# B&R Automation Studio project Embraco_LinkaNaOdlievanieRotorov_DokoncovaciaStanica_Rev2 (part 4)

#### OvladanieGripra.st
```iecst
ACTION OvladanieGripra:

	//Volanie funkcie SequenceControl//
	SequenceControl(SC:= SC_OvlGripra);

	CASE SC_OvlGripra.Step OF

		0:
			SC_OvlGripra.StepName:= '0 - Nulovanie';
			Otvor_Griper:= FALSE;
			Zatvor_Griper:= FALSE;
			doValcovanie_GriperOTVOR:= FALSE;
			doValcovanie_GriperZATVOR:= FALSE;
			IF SC_Valcovanie.Step <> 0 THEN
				SC_OvlGripra.ResetStep:= TRUE;
				SC_OvlGripra.Step:= 1;
			END_IF

		1:
			SC_OvlGripra.StepName:= '1 - Rozhodnutie o cinnosti';
			IF Otvor_Griper THEN
				SC_OvlGripra.Step:= 10;
			ELSIF Zatvor_Griper THEN
				SC_OvlGripra.Step:= 20;
			END_IF

		10:
			SC_OvlGripra.StepName:= '10 - Otvorenie gripra';
			SC_OvlGripra.IdleTime.PT:= T#3s;
			SC_OvlGripra.AlarmTime.PT:= T#3s;

			IF Valcovanie_Manual THEN
				SC_OvlGripra.IdleTime.IN:= TRUE;
			ELSE
				SC_OvlGripra.AlarmTime.IN:= TRUE;
			END_IF

			IF NOT SC_OvlGripra.Switch1 THEN
				doValcovanie_GriperOTVOR:= TRUE;
				SC_OvlGripra.Switch1:= TRUE;
			END_IF

			IF SC_OvlGripra.AlarmTime.Q THEN
				Alarmy[63]:= TRUE;
				PoruchaStanicaValcovania:= TRUE;
			END_IF

			IF diValcovanie_GriperOtvoreny OR SC_OvlGripra.IdleTime.Q THEN
				SC_OvlGripra.ResetStep:= TRUE;
				SC_OvlGripra.Step:= 0;
			END_IF

		20:
			SC_OvlGripra.StepName:= '20 - Zatvorenie gripra';
			SC_OvlGripra.IdleTime.PT:= T#3s;
			SC_OvlGripra.AlarmTime.PT:= T#3s;

			IF Valcovanie_Manual THEN
				SC_OvlGripra.IdleTime.IN:= TRUE;
			ELSE
				SC_OvlGripra.AlarmTime.IN:= TRUE;
			END_IF

			IF NOT SC_OvlGripra.Switch1 THEN
				doValcovanie_GriperZATVOR:= TRUE;
				SC_OvlGripra.Switch1:= TRUE;
			END_IF

			IF SC_OvlGripra.AlarmTime.Q THEN
				Alarmy[62]:= TRUE;
				PoruchaStanicaValcovania:= TRUE;
			END_IF

			IF diValcovanie_GriperZatvoreny OR SC_OvlGripra.IdleTime.Q THEN
				SC_OvlGripra.ResetStep:= TRUE;
				SC_OvlGripra.Step:= 0;
			END_IF

	END_CASE

			END_ACTION
```

#### OvladanieZdvihuRotora.st
```iecst
ACTION OvladanieZdvihuRotora:

	//Volanie funkcie SequenceControl//
	SequenceControl(SC:= SC_OvlZdvihu);

	CASE SC_OvlZdvihu.Step OF

		0:
			SC_OvlZdvihu.StepName:= '0 - Nulovanie';
			Rotor_ZDVIHNI:= FALSE;
			Rotor_POLOZ:= FALSE;
			doValcovanie_ZDVIH_Rotora:= FALSE;
			doValcovanie_ZOSTUP_Rotora:= FALSE;
			IF SC_Valcovanie.Step <> 0 THEN
				SC_OvlZdvihu.ResetStep:= TRUE;
				SC_OvlZdvihu.Step:= 1;
			END_IF

		1:
			SC_OvlZdvihu.StepName:= '1 - Rozhodnutie o cinnosti';
			IF Rotor_ZDVIHNI THEN
				SC_OvlZdvihu.Step:= 10;
			ELSIF Rotor_POLOZ THEN
				SC_OvlZdvihu.Step:= 20;
			END_IF

		10:
			SC_OvlZdvihu.StepName:= '10 - Zodvihnutie rotora';
			SC_OvlZdvihu.IdleTime.PT:= T#3s;
			SC_OvlZdvihu.AlarmTime.PT:= T#3s;

			IF Valcovanie_Manual THEN
				SC_OvlZdvihu.IdleTime.IN:= TRUE;
			ELSE
				SC_OvlZdvihu.AlarmTime.IN:= TRUE;
			END_IF

			IF NOT SC_OvlZdvihu.Switch1 THEN
				doValcovanie_ZDVIH_Rotora:= TRUE;
				SC_OvlZdvihu.Switch1:= TRUE;
			END_IF

			IF SC_OvlZdvihu.AlarmTime.Q THEN
				Alarmy[60]:= TRUE;
				PoruchaStanicaValcovania:= TRUE;
			END_IF

			IF diValcovanie_ZdvihHornaPoloha OR SC_OvlZdvihu.IdleTime.Q THEN
				SC_OvlZdvihu.ResetStep:= TRUE;
				SC_OvlZdvihu.Step:= 0;
			END_IF

		20:
			SC_OvlZdvihu.StepName:= '20 - Polozenie rotora';
			SC_OvlZdvihu.IdleTime.PT:= T#3s;
			SC_OvlZdvihu.AlarmTime.PT:= T#3s;

			IF Valcovanie_Manual THEN
				SC_OvlZdvihu.IdleTime.IN:= TRUE;
			ELSE
				SC_OvlZdvihu.AlarmTime.IN:= TRUE;
			END_IF

			IF NOT SC_OvlZdvihu.Switch1 THEN
				doValcovanie_ZOSTUP_Rotora:= TRUE;
				SC_OvlZdvihu.Switch1:= TRUE;
			END_IF

			IF SC_OvlZdvihu.AlarmTime.Q THEN
				Alarmy[61]:= TRUE;
				PoruchaStanicaValcovania:= TRUE;
			END_IF

			IF diValcovanie_ZdvihSpodnaPoloha OR SC_OvlZdvihu.IdleTime.Q THEN
				SC_OvlZdvihu.ResetStep:= TRUE;
				SC_OvlZdvihu.Step:= 0;
			END_IF

	END_CASE

			END_ACTION
```

#### OvladanieOtacaniaRotora.st
```iecst
ACTION OvladanieOtacaniaRotora:

	//Zadanie rýchlosti otáčania rotora//
	Valcovanie_FM_RychlostOtac_Hz:= TP_Valcovanie_RychlostOtacania;

	//Volanie funkcie SequenceControl//
	SequenceControl(SC:= SC_OvlOtacania);

	CASE SC_OvlOtacania.Step OF

		0:
			SC_OvlOtacania.StepName:= '0 - Nulovanie';
			FM_Menic[2].Input.Command.RunForward:= FALSE;
			FM_Menic[2].Input.Command.RunBackward:= FALSE;
			RotorOtacaj_VPRED:= FALSE;
			RotorOtacaj_VZAD:= FALSE;
			IF SC_Valcovanie.Step <> 0 THEN
				SC_OvlOtacania.ResetStep:= TRUE;
				SC_OvlOtacania.Step:= 1;
			END_IF

		1:
			SC_OvlOtacania.StepName:= '1 - Rozhodnutie o cinnosti';
			IF RotorOtacaj_VPRED THEN
				SC_OvlOtacania.Step:= 10;
			ELSIF RotorOtacaj_VZAD THEN
				SC_OvlOtacania.Step:= 20;
			END_IF

		10:
			SC_OvlOtacania.StepName:= '10 - Otacanie rotora VPRED';
			SC_OvlOtacania.IdleTime.PT:= T#5s;
			SC_OvlOtacania.AlarmTime.PT:= T#15s;
			FM_Menic[2].Input.HighSpeed:= (Valcovanie_FM_RychlostOtac_Hz * 10); //v Hz
			FM_Menic[2].Input.AccTime:= 1;  //0.1s
			FM_Menic[2].Input.DecTime:= 1;  //0.1s
			RotorOtacaj_VZAD:= FALSE;

			IF NOT SC_OvlOtacania.Switch1 THEN
				FM_Menic[2].Input.Command.RunForward:= TRUE;
				SC_OvlOtacania.Switch1:= TRUE;
			END_IF

			IF NOT RotorOtacaj_VPRED THEN
				SC_OvlOtacania.ResetStep:= TRUE;
				SC_OvlOtacania.Step:= 0;
			END_IF

		20:
			SC_OvlOtacania.StepName:= '20 - Otacanie rotora VZAD';
			SC_OvlOtacania.IdleTime.PT:= T#5s;
			SC_OvlOtacania.AlarmTime.PT:= T#15s;
			FM_Menic[2].Input.HighSpeed:= (Valcovanie_FM_RychlostOtac_Hz * 10); //v Hz
			FM_Menic[2].Input.AccTime:= 1;  //0.1s
			FM_Menic[2].Input.DecTime:= 1;  //0.1s
			RotorOtacaj_VPRED:= FALSE;

			IF NOT SC_OvlOtacania.Switch1 THEN
				FM_Menic[2].Input.Command.RunBackward:= TRUE;
				SC_OvlOtacania.Switch1:= TRUE;
			END_IF

			IF NOT RotorOtacaj_VZAD THEN
				SC_OvlOtacania.ResetStep:= TRUE;
				SC_OvlOtacania.Step:= 0;
			END_IF

	END_CASE

END_ACTION
```

### Program Logical/Program/StanicaVonkajsiehoValcovania (IEC)

#### Main.st - Init, cyclic, exit code
```iecst
PROGRAM _INIT
	(* Insert code here *)

END_PROGRAM

PROGRAM _CYCLIC

	//Volanie podprogramov//
	OvlHornehoPritlaku;
	OvlOtacaniaNastroja;
	OvlZdvihuRotora;

	//Volanie funkcie SequenceControl//
	SequenceControl(SC:= SC_Valcovanie2);

	Valcovanie2_CasStrekuOleja_s;
	Valcovanie2_CasValcovania_s;

	//***************************Dávka oleja**********************************//
	IF Valcovanie2_DavkaOleja THEN
		doValc2_DavkaOleja:= TRUE;
		CasDavkyOleja.IN:= TRUE;
	END_IF

	IF CasDavkyOleja.Q THEN
		Valcovanie2_DavkaOleja:= FALSE;
		CasDavkyOleja.IN:= FALSE;
		doValc2_DavkaOleja:= FALSE;
	END_IF

	CasDavkyOleja.PT:= REAL_TO_TIME(Valcovanie2_CasStrekuOleja_s * 1000);
	CasDavkyOleja();

	//Reset sekcie //
	IF Valcovanie2_Reset OR NOT BezpOkruhOplotenia_Aktivovany OR PoruchaStanicaValcovania2 THEN
		SC_Valcovanie2.Step:= 0;
	END_IF

	CASE SC_Valcovanie2.Step OF

		0:
			SC_Valcovanie2.StepName:='0 - Nulovanie';
			SC_OvlHornehoPritlaku.Step:= 0;
			SC_OvlOtacaniaNastroja.Step:= 0;
			SC_OvlZdvihuRotora.Step:= 0;
			Valcovanie2_Automat:= FALSE;
			Valcovanie2_KoniecVyroby:= FALSE;
			Valcovanie2_KoniecCyklu:= FALSE;
			Valcovanie2_Manual:= FALSE;
			Valcovanie2_PoINIT:= FALSE;
			Valcovanie2_Reset:= FALSE;
			Valcovanie2_ZdvihVPOZICI:= FALSE;
			Valcovanie2_UkoncilCyklus:= FALSE;
			RR_ZdvihRotora_PozValcovania:= FALSE;
			RR_ZdvihRotora_PozVychodzia:= FALSE;
			PocetCyklovValcovania:= 0;
			Priznak_ValcovanieNG:= FALSE;
			Priznak_ValcovanieOK:= FALSE;
			IF BezpOkruhOplotenia_Aktivovany AND NOT PoruchaStanicaValcovania2 THEN
				SC_Valcovanie2.ResetStep:= TRUE;
				SC_Valcovanie2.Step:= 1;
			END_IF

		1:
			SC_Valcovanie2.StepName:='1 - Rozhodnutie o cinnosti';
			IF Valcovanie2_Automat THEN
				SC_Valcovanie2.Step:= 2;
			ELSIF Valcovanie2_Manual THEN
				SC_Valcovanie2.Step:= 700;
			END_IF

			//********************************************************Inicializácia****************************************************************************//

		2:
			SC_Valcovanie2.StepName:='2 - Inicializacia - cakanie na spustenie';
			SC_Valcovanie2.IdleTime.PT:= T#500ms;
			SC_Valcovanie2.AlarmTime.PT:= T#5s;
			SC_Valcovanie2.IdleTime.IN:= TRUE;

			IF SC_Valcovanie2.IdleTime.Q AND diStol_SnimacPolohyStola THEN
				SC_Valcovanie2.ResetStep:= TRUE;
				SC_Valcovanie2.Step:= 4;
			END_IF

		4:
			SC_Valcovanie2.StepName:='4 - Inicializacia - kontrola home serva zdvihu rotora';
			SC_Valcovanie2.IdleTime.PT:= T#500ms;
			SC_Valcovanie2.AlarmTime.PT:= T#5s;

			IF Motion[4].status.DriveStatus.HomingOk THEN
				SC_Valcovanie2.ResetStep:= TRUE;
				SC_Valcovanie2.Step:= 6;
			ELSE
				SC_Valcovanie2.ResetStep:= TRUE;
				SC_Valcovanie2.Step:= 5;
			END_IF

		5:
			SC_Valcovanie2.StepName:='5 - Inicializacia - homing serva zdvihu rotora';
			SC_Valcovanie2.IdleTime.PT:= T#500ms;
			SC_Valcovanie2.AlarmTime.PT:= T#5s;

			IF NOT SC_Valcovanie2.Switch1 THEN
				ZdvihRotora_HOME:= TRUE;
				SC_Valcovanie2.Switch1:= TRUE;
			END_IF

			IF Motion[4].status.DriveStatus.HomingOk THEN
				SC_Valcovanie2.IdleTime.IN:= TRUE;
			END_IF

			IF Motion[4].status.DriveStatus.HomingOk AND SC_Valcovanie2.IdleTime.Q AND Motion[4].state.StandStill THEN
				SC_Valcovanie2.ResetStep:= TRUE;
				SC_Valcovanie2.Step:= 6;
			END_IF

		6:
			SC_Valcovanie2.StepName:='6 - Inicializacia - zasunutie zdvihu rotora do vychodiskovej pozicie';
			SC_Valcovanie2.IdleTime.PT:= T#500ms;
			SC_Valcovanie2.AlarmTime.PT:= T#5s;

			IF NOT SC_Valcovanie2.Switch1 AND (Valcovanie2_AktualPozMM <> Valcovanie2_ZadanaPozSTART_MM) AND SC_OvlZdvihuRotora.Step = 1 THEN
				ZdvihRotora_PoziciaSTART:= TRUE;
				SC_Valcovanie2.Switch1:= TRUE;
			END_IF

			IF (Valcovanie2_AktualPozMM = Valcovanie2_ZadanaPozSTART_MM) AND Motion[4].state.StandStill THEN
				SC_Valcovanie2.ResetStep:= TRUE;
				SC_Valcovanie2.Step:= 9;
			END_IF

		9:
			SC_Valcovanie2.StepName:='9 - Inicializacia - vysunutie horneho pritlaku dole';
			SC_Valcovanie2.IdleTime.PT:= T#4s;
			SC_Valcovanie2.AlarmTime.PT:= T#5s;

			IF NOT SC_Valcovanie2.Switch1 AND SC_OvlHornehoPritlaku.Step = 1 THEN
				HornyPritlak_DOLE:= TRUE;
				SC_Valcovanie2.Switch1:= TRUE;
			END_IF

			IF diValc2_PritlakVysunuty THEN
				SC_Valcovanie2.ResetStep:= TRUE;
				SC_Valcovanie2.Step:= 10;
			END_IF

		10:
			SC_Valcovanie2.StepName:='10 - Inicializacia - spustenie otacania nastroja';
			SC_Valcovanie2.IdleTime.PT:= T#4s;
			SC_Valcovanie2.AlarmTime.PT:= T#5s;

			IF NOT SC_Valcovanie2.Switch1 AND SC_OvlOtacaniaNastroja.Step = 1 AND VonkajsieValcovanie_AKTIVNE THEN
				OtacanieNastroja_VPRED:= TRUE;
				SC_Valcovanie2.IdleTime.IN:= TRUE;
				SC_Valcovanie2.Switch1:= TRUE;
			END_IF

			IF SC_Valcovanie2.IdleTime.Q OR NOT VonkajsieValcovanie_AKTIVNE THEN
				Valcovanie2_PoINIT:= TRUE;
				SC_Valcovanie2.ResetStep:= TRUE;
				SC_Valcovanie2.Step:= 100;
			END_IF

			//********************************************************Automatický režim****************************************************************************//
		100:
			SC_Valcovanie2.StepName:='100 - Automaticky rezim - cakanie na start cyklu';
			SC_Valcovanie2.IdleTime.PT:= T#500ms;
			SC_Valcovanie2.AlarmTime.PT:= T#5s;

            SC_Valcovanie2.IdleTime.IN:= NOT diValc2_PritomnostRotora;

			IF Valcovanie2_KoniecCyklu THEN
				SC_Valcovanie2.ResetStep:= TRUE;
				SC_Valcovanie2.Step:= 105;
			ELSIF NOT VonkajsieValcovanie_AKTIVNE THEN
				SC_Valcovanie2.ResetStep:= TRUE;
				SC_Valcovanie2.Step:= 120;
			ELSIF Stol_PoINIT AND NOT Valcovanie2_UkoncilCyklus AND diValc2_PritomnostRotora AND diStol_SnimacPolohyStola THEN
				SC_Valcovanie2.ResetStep:= TRUE;
				SC_Valcovanie2.Step:= 101;
			ELSIF Stol_PoINIT AND NOT Valcovanie2_UkoncilCyklus AND NOT diValc2_PritomnostRotora AND SC_Valcovanie2.IdleTime.Q THEN
				SC_Valcovanie2.ResetStep:= TRUE;
				SC_Valcovanie2.Step:= 120;
			ELSIF Valcovanie2_KoniecVyroby AND NOT Stol_Automat THEN
				SC_Valcovanie2.ResetStep:= TRUE;
				SC_Valcovanie2.Step:= 105;
			END_IF

		101:
			SC_Valcovanie2.StepName:='101 - Automaticky rezim - zdvih rotora, streknutie oleja';
			SC_Valcovanie2.IdleTime.PT:= T#500ms;
			SC_Valcovanie2.AlarmTime.PT:= T#5s;

			IF NOT SC_Valcovanie2.Switch1 AND SC_OvlZdvihuRotora.Step = 1 THEN
				ZdvihRotora_VALCOVANIE:= TRUE;
				SC_Valcovanie2.Switch1:= TRUE;
			END_IF

			IF Priznak_ValcovanieOK AND Valcovanie2_AktualPozMM = 13 AND Motion[4].state.StandStill AND diValc2_PritomnostRotora AND NOT diValc2_SpomalenieZdvihu THEN
				Priznak_ValcovanieOK:= FALSE;
				SC_Valcovanie2.ResetStep:= TRUE;
				SC_Valcovanie2.Step:= 120;
			ELSIF Priznak_ValcovanieOK AND Valcovanie2_AktualPozMM = 13 AND Motion[4].state.StandStill AND (NOT diValc2_PritomnostRotora OR diValc2_SpomalenieZdvihu) THEN
				Alarmy[74]:= TRUE;
				PoruchaStanicaValcovania2:= TRUE;
			ELSIF Priznak_ValcovanieNG AND (Valcovanie2_AktualPozMM = 13) AND Motion[4].state.StandStill THEN
				SC_Valcovanie2.ResetStep:= TRUE;
				SC_Valcovanie2.Step:= 110;
			END_IF

		105:
			SC_Valcovanie2.StepName:='105 - Automaticky rezim - zdvih vrchneho pritlaku';
			SC_Valcovanie2.IdleTime.PT:= T#500ms;
			SC_Valcovanie2.AlarmTime.PT:= T#5s;

			IF NOT SC_Valcovanie2.Switch1 THEN
				HornyPritlak_HORE:= TRUE;
			END_IF

			IF diValc2_PritlakZasunuty THEN
				SC_Valcovanie2.ResetStep:= TRUE;
				SC_Valcovanie2.Step:= 0;
			END_IF

		110:
			SC_Valcovanie2.StepName:='110 - Automaticky rezim - zdvih vrchneho pritlaku po NG kusu';
			SC_Valcovanie2.IdleTime.PT:= T#500ms;
			SC_Valcovanie2.AlarmTime.PT:= T#5s;

			IF NOT SC_Valcovanie2.Switch1 THEN
				HornyPritlak_HORE:= TRUE;
			END_IF

			IF diValc2_PritlakZasunuty THEN
				Alarmy[75]:= TRUE;
				PoruchaStanicaValcovania2:= TRUE;
			END_IF

		120:
			SC_Valcovanie2.StepName:='120 - Automaticky rezim - vystavenie signalu ukoncenie pracovneho cyklu';
			SC_Valcovanie2.IdleTime.PT:= T#500ms;
			SC_Valcovanie2.AlarmTime.PT:= T#5s;

			Valcovanie2_UkoncilCyklus:= TRUE;
			SC_Valcovanie2.ResetStep:= TRUE;
			SC_Valcovanie2.Step:= 121;

		121:
			SC_Valcovanie2.StepName:='121 - Automaticky rezim - cakanie na otocenie stola';
			SC_Valcovanie2.IdleTime.PT:= T#500ms;
			SC_Valcovanie2.AlarmTime.PT:= T#5s;

			IF NOT Valcovanie2_UkoncilCyklus THEN
				SC_Valcovanie2.ResetStep:= TRUE;
				SC_Valcovanie2.Step:= 100;
			ELSIF Valcovanie2_KoniecVyroby AND NOT Stol_Automat THEN
				SC_Valcovanie2.ResetStep:= TRUE;
				SC_Valcovanie2.Step:= 105;
			ELSIF Valcovanie2_KoniecCyklu THEN
				SC_Valcovanie2.ResetStep:= TRUE;
				SC_Valcovanie2.Step:= 105;
			END_IF

			//********************************************************Ručný režim***********************************************************************************//
		700:
			SC_Valcovanie2.StepName:='700 - Rucny rezim';

	END_CASE

				END_PROGRAM

PROGRAM _EXIT
				(* Insert code here *)

				END_PROGRAM
```

#### Variables.var - Local variables
```iecst
VAR
	SC_OvlZdvihuRotora : SequenceControlTyp;
	ZdvihRotora_JoggHORE : BOOL;
	ZdvihRotora_JoggDOLE : BOOL;
	ZdvihRotora_VALCOVANIE : BOOL;
	ZdvihRotora_HOME : BOOL;
	ZdvihRotora_PoziciaSTART : BOOL;
	ZdvihRotora_PoziciaVALCOVANIA : BOOL;
	SC_OvlOtacaniaNastroja : SequenceControlTyp;
	OtacanieNastroja_VPRED : BOOL;
	OtacanieNastroja_VZAD : BOOL;
	SC_OvlHornehoPritlaku : SequenceControlTyp;
	HornyPritlak_HORE : BOOL;
	HornyPritlak_DOLE : BOOL;
	CasDavkyOleja : TON;
	RR_ZdvihRotora_PozVychodzia : BOOL;
	RR_ZdvihRotora_PozValcovania : BOOL;
	PocetCyklovValcovania : USINT;
	Priznak_ValcovanieNG : BOOL;
	Priznak_ValcovanieOK : BOOL;
	TaktTime : TON;
	NameranyTaktime : TIME;
END_VAR
```

#### OvlZdvihuRotora.st
```iecst
ACTION OvlZdvihuRotora:

	//Parametre zdvihu rotora//
	Valcovanie2_ServoJoggRychl_MM_s;
	Valcovanie2_ServoPracRychl1_MM_s; //Rýchlost priblíženia
	Valcovanie2_ServoPracRychl2_MM_s; //Rýchlosť valcovania
	Valcovanie2_FM_RozbehRampa_s;
	Valcovanie2_FM_DobehRampa_s;
	Valcovanie2_MomentPritlaku_Nm:= 3; //3Nm

	//Volanie funkcie SequenceControl//
	SequenceControl(SC:= SC_OvlZdvihuRotora);

	CASE SC_OvlZdvihuRotora.Step OF

		0:
			SC_OvlZdvihuRotora.StepName:= '0 - Nulovanie';
			ZdvihRotora_JoggDOLE:= FALSE;
			ZdvihRotora_JoggHORE:= FALSE;
			ZdvihRotora_HOME:= FALSE;
			ZdvihRotora_VALCOVANIE:= FALSE;
			ZdvihRotora_PoziciaSTART:= FALSE;
			ZdvihRotora_PoziciaVALCOVANIA:= FALSE;
			Motion[4].cmd.home:= FALSE;
			Motion[4].cmd.moveAbsolute:= FALSE;
			Motion[4].cmd.moveJogNeg:= FALSE;
			Motion[4].cmd.moveJogPos:= FALSE;
			Motion[4].cmd.moveVelocity:= FALSE;
			Valcovanie2_PrebiehaHoming:= FALSE;
			Motion[4].par.direction:= 0;

			IF SC_Valcovanie2.Step <> 0 AND (NOT Motion[4].status.DriveStatus.HomingOk OR Motion[4].state.StandStill) THEN
				Motion[4].cmd.halt:= FALSE;
				SC_OvlZdvihuRotora.ResetStep:= TRUE;
				SC_OvlZdvihuRotora.Step:= 1;
			END_IF

		1:
			SC_OvlZdvihuRotora.StepName:= '1 - Rozhodnutie o cinnosti';
			IF ZdvihRotora_JoggDOLE THEN
				SC_OvlZdvihuRotora.Step:= 10;
			ELSIF ZdvihRotora_JoggHORE THEN
				SC_OvlZdvihuRotora.Step:= 20;
			ELSIF ZdvihRotora_HOME THEN
				SC_OvlZdvihuRotora.Step:= 30;
			ELSIF ZdvihRotora_VALCOVANIE THEN
				SC_OvlZdvihuRotora.Step:= 40;
			ELSIF ZdvihRotora_PoziciaSTART THEN
				SC_OvlZdvihuRotora.Step:= 50;
			ELSIF ZdvihRotora_PoziciaVALCOVANIA THEN
				SC_OvlZdvihuRotora.Step:= 60;
			END_IF

		10:
			SC_OvlZdvihuRotora.StepName:= '10 - Jogging DOLE';
			SC_OvlZdvihuRotora.IdleTime.PT:= T#3s;
			SC_OvlZdvihuRotora.AlarmTime.PT:= T#3s;

			Motion[4].par.velocityJog:= (Valcovanie2_ServoJoggRychl_MM_s * 100);
			Motion[4].par.acc := (Valcovanie2_ServoJoggRychl_MM_s * 1000);
			Motion[4].par.dec := (Valcovanie2_ServoJoggRychl_MM_s * 1000);

			IF NOT SC_OvlZdvihuRotora.Switch1 THEN
				Motion[4].cmd.moveJogNeg:= TRUE;
				SC_OvlZdvihuRotora.Switch1:= TRUE;
			END_IF

			IF (NOT ZdvihRotora_JoggDOLE OR Valcovanie2_AktualPozMM <= 13)THEN
				Motion[4].cmd.moveJogNeg:= FALSE;
				SC_OvlZdvihuRotora.ResetStep:= TRUE;
				SC_OvlZdvihuRotora.Step:= 0;
			END_IF

			IF diValc2_ZdvihSpodnyLimit THEN
				Motion[4].cmd.halt:= TRUE;
				Alarmy[56]:= TRUE;
				PoruchaStanicaValcovania2:= TRUE;
			END_IF

		20:
			SC_OvlZdvihuRotora.StepName:= '20 - Jogging HORE';
			SC_OvlZdvihuRotora.IdleTime.PT:= T#3s;
			SC_OvlZdvihuRotora.AlarmTime.PT:= T#3s;

			Motion[4].par.velocityJog:= (Valcovanie2_ServoJoggRychl_MM_s * 100);
			Motion[4].par.acc := (Valcovanie2_ServoJoggRychl_MM_s * 1000);
			Motion[4].par.dec := (Valcovanie2_ServoJoggRychl_MM_s * 1000);

			IF NOT SC_OvlZdvihuRotora.Switch1 THEN
				Motion[4].cmd.moveJogPos:= TRUE;
				SC_OvlZdvihuRotora.Switch1:= TRUE;
			END_IF

			IF (NOT ZdvihRotora_JoggHORE OR Valcovanie2_AktualPozMM >= 185)THEN
				Motion[4].cmd.moveJogPos:= FALSE;
				SC_OvlZdvihuRotora.ResetStep:= TRUE;
				SC_OvlZdvihuRotora.Step:= 0;
			END_IF

			IF diValc2_ZdvihHornyLimit THEN
				Motion[4].cmd.halt:= TRUE;
				Alarmy[56]:= TRUE;
				PoruchaStanicaValcovania2:= TRUE;
			END_IF

		30:
			SC_OvlZdvihuRotora.StepName:= '30 - Start homingu';
			SC_OvlZdvihuRotora.IdleTime.PT:= T#500ms;
			SC_OvlZdvihuRotora.AlarmTime.PT:= T#3s;

			IF NOT SC_OvlZdvihuRotora.Switch1 THEN
				Motion[4].cmd.home:= TRUE;
				Valcovanie2_PrebiehaHoming:= TRUE;
				SC_OvlZdvihuRotora.IdleTime.IN:= TRUE;
				SC_OvlZdvihuRotora.Switch1:= TRUE;
			END_IF

			IF SC_OvlZdvihuRotora.IdleTime.Q THEN
				SC_OvlZdvihuRotora.ResetStep:= TRUE;
				SC_OvlZdvihuRotora.Step:= 31;
			END_IF

		31:
			SC_OvlZdvihuRotora.StepName:= '31 - Ukoncenie homingu';
			SC_OvlZdvihuRotora.IdleTime.PT:= T#3s;
			SC_OvlZdvihuRotora.AlarmTime.PT:= T#3s;

			IF Valcovanie2_HomingOK AND Motion[4].state.StandStill THEN
				SC_OvlZdvihuRotora.ResetStep:= TRUE;
				SC_OvlZdvihuRotora.Step:= 0;
			END_IF

		40:
			SC_OvlZdvihuRotora.StepName:= '40 - Valcovanie,chod rychlo na spomalovaci snimac';
			SC_OvlZdvihuRotora.IdleTime.PT:= T#3s;
			SC_OvlZdvihuRotora.AlarmTime.PT:= T#3s;

			Motion[4].par.velocity:= (Valcovanie2_ServoPracRychl1_MM_s * 100);
			Motion[4].par.acc := (Valcovanie2_ServoPracRychl1_MM_s * 1000);
			Motion[4].par.dec := (Valcovanie2_ServoPracRychl1_MM_s * 1000);
			Motion[4].par.direction:= 0;

			IF NOT SC_OvlZdvihuRotora.Switch1 THEN
				Motion[4].cmd.moveVelocity:= TRUE;
				PocetCyklovValcovania:= PocetCyklovValcovania + 1;
				TaktTime.IN:= TRUE;
				SC_OvlZdvihuRotora.Switch1:= TRUE;
			END_IF

			IF EDGEPOS(diValc2_SpomalenieZdvihu) THEN
				SC_OvlZdvihuRotora.ResetStep:= TRUE;
				SC_OvlZdvihuRotora.Step:= 41;
			ELSIF Valcovanie2_AktualPozMM >= 118 THEN
				SC_OvlZdvihuRotora.ResetStep:= TRUE;
				SC_OvlZdvihuRotora.Step:= 41;
			ELSIF diValc2_ZdvihHornyLimit THEN
				Motion[4].cmd.halt:= TRUE;
				Alarmy[56]:= TRUE;
				PoruchaStanicaValcovania2:= TRUE;
			END_IF

		41:
			SC_OvlZdvihuRotora.StepName:= '41 - Valcovanie,chod pomaly na poziciu';
			SC_OvlZdvihuRotora.IdleTime.PT:= T#1s;
			SC_OvlZdvihuRotora.AlarmTime.PT:= T#3s;

			Motion[4].par.velocity:= (Valcovanie2_ServoPracRychl2_MM_s * 100);
			Motion[4].par.acc := (Valcovanie2_ServoPracRychl2_MM_s * 1000);
			Motion[4].par.dec := (Valcovanie2_ServoPracRychl2_MM_s * 1000);
			Motion[4].par.position:= (Valcovanie2_ZadanaPozMM * 100); //180mm

			IF NOT SC_OvlZdvihuRotora.Switch1 THEN
				Motion[4].cmd.moveAbsolute:= TRUE;
				IF PocetCyklovValcovania >= Valcovanie2_PocetCyklStrekuOleja THEN
					Valcovanie2_DavkaOleja:= TRUE;
					PocetCyklovValcovania:= 0;
				END_IF
				SC_OvlZdvihuRotora.Switch1:= TRUE;
			END_IF

			IF (Valcovanie2_AktualPozMM = Valcovanie2_ZadanaPozMM) AND Motion[4].state.StandStill THEN
				SC_OvlZdvihuRotora.ResetStep:= TRUE;
				SC_OvlZdvihuRotora.Step:= 45;
			ELSIF Motion[4].status.ActTorque >= 20 THEN
				Motion[4].cmd.halt:= TRUE;
				Priznak_ValcovanieNG:= TRUE;
				SC_OvlZdvihuRotora.ResetStep:= TRUE;
				SC_OvlZdvihuRotora.Step:= 42;
			ELSIF diValc2_ZdvihHornyLimit THEN
				Motion[4].cmd.halt:= TRUE;
				Alarmy[56]:= TRUE;
				PoruchaStanicaValcovania2:= TRUE;
			END_IF

		42:
			SC_OvlZdvihuRotora.StepName:= '42 - Valcovanie,zastavenie po dosiahnutí momentu';
			SC_OvlZdvihuRotora.IdleTime.PT:= T#1s;
			SC_OvlZdvihuRotora.AlarmTime.PT:= T#3s;
			SC_OvlZdvihuRotora.IdleTime.IN:= TRUE;

			IF NOT Motion[4].cmd.halt THEN
				SC_OvlZdvihuRotora.ResetStep:= TRUE;
				SC_OvlZdvihuRotora.Step:= 45;
			END_IF

			IF SC_OvlZdvihuRotora.IdleTime.Q THEN
				Motion[4].cmd.halt:= FALSE;
			END_IF

		45:
			SC_OvlZdvihuRotora.StepName:= '45 - Valcovanie,chod pomalou rychlostou dole';
			SC_OvlZdvihuRotora.IdleTime.PT:= T#50ms;
			SC_OvlZdvihuRotora.AlarmTime.PT:= T#3s;
			SC_OvlZdvihuRotora.IdleTime.IN:= TRUE;

			Motion[4].par.velocity:= (Valcovanie2_ServoPracRychl1_MM_s * 100);
			Motion[4].par.acc := (Valcovanie2_ServoPracRychl1_MM_s * 1000);
			Motion[4].par.dec := (Valcovanie2_ServoPracRychl1_MM_s * 1000);
			Motion[4].par.direction:= 1;

			IF NOT SC_OvlZdvihuRotora.Switch1 AND SC_OvlZdvihuRotora.IdleTime.Q THEN
				Motion[4].cmd.moveVelocity:= TRUE;
				SC_OvlZdvihuRotora.Switch1:= TRUE;
			END_IF

			IF NOT diValc2_SpomalenieZdvihu AND Valcovanie2_AktualPozMM < 118 THEN
				SC_OvlZdvihuRotora.ResetStep:= TRUE;
				SC_OvlZdvihuRotora.Step:= 46;
			ELSIF Valcovanie2_AktualPozMM <= 95 THEN
				SC_OvlZdvihuRotora.ResetStep:= TRUE;
				SC_OvlZdvihuRotora.Step:= 46;
			ELSIF diValc2_ZdvihSpodnyLimit THEN
				Motion[4].cmd.halt:= TRUE;
				Alarmy[56]:= TRUE;
				PoruchaStanicaValcovania2:= TRUE;
			END_IF

		46:
			SC_OvlZdvihuRotora.StepName:= '46 - Valcovanie, chod rychlo do vychodiskovej pozicie';
			SC_OvlZdvihuRotora.IdleTime.PT:= T#3s;
			SC_OvlZdvihuRotora.AlarmTime.PT:= T#3s;

			Motion[4].par.velocity:= (Valcovanie2_ServoPracRychl1_MM_s * 100);
			Motion[4].par.acc := (Valcovanie2_ServoPracRychl1_MM_s * 1000);
			Motion[4].par.dec := (Valcovanie2_ServoPracRychl1_MM_s * 1000);
			Motion[4].par.position:= 1300; //13mm

			IF NOT SC_OvlZdvihuRotora.Switch1 THEN
				Motion[4].cmd.moveAbsolute:= TRUE;
				SC_OvlZdvihuRotora.Switch1:= TRUE;
			END_IF

			IF (Valcovanie2_AktualPozMM = 13) AND Motion[4].state.StandStill AND NOT Priznak_ValcovanieNG THEN
				Priznak_ValcovanieOK:= TRUE;
				NameranyTaktime:= TaktTime.ET;
				TaktTime.IN:= FALSE;
				SC_OvlZdvihuRotora.ResetStep:= TRUE;
				SC_OvlZdvihuRotora.Step:= 0;
			ELSIF diValc2_ZdvihSpodnyLimit THEN
				Motion[4].cmd.halt:= TRUE;
				Alarmy[56]:= TRUE;
				PoruchaStanicaValcovania2:= TRUE;
			END_IF

		50:
			SC_OvlZdvihuRotora.StepName:= '50 - Presun do pozicie START';
			SC_OvlZdvihuRotora.IdleTime.PT:= T#3s;
			SC_OvlZdvihuRotora.AlarmTime.PT:= T#3s;

			Motion[4].par.velocity:= (Valcovanie2_ServoPracRychl1_MM_s * 100);
			Motion[4].par.acc := (Valcovanie2_ServoPracRychl1_MM_s * 1000);
			Motion[4].par.dec := (Valcovanie2_ServoPracRychl1_MM_s * 1000);
			Motion[4].par.position:= 1300; //13mm

			IF NOT SC_OvlZdvihuRotora.Switch1 THEN
				Motion[4].cmd.moveAbsolute:= TRUE;
				SC_OvlZdvihuRotora.Switch1:= TRUE;
			END_IF

			IF (Valcovanie2_AktualPozMM = 13) AND Motion[4].state.StandStill THEN
				Valcovanie2_ZdvihVPOZICI:= TRUE;
				SC_OvlZdvihuRotora.ResetStep:= TRUE;
				SC_OvlZdvihuRotora.Step:= 0;
			ELSIF diValc2_ZdvihSpodnyLimit THEN
				Motion[4].cmd.halt:= TRUE;
				Alarmy[56]:= TRUE;
				PoruchaStanicaValcovania2:= TRUE;
			END_IF

		60:
			SC_OvlZdvihuRotora.StepName:= '60 - Presun do pozicie VALCOVANIA';
			SC_OvlZdvihuRotora.IdleTime.PT:= T#3s;
			SC_OvlZdvihuRotora.AlarmTime.PT:= T#3s;

			Motion[4].par.velocity:= (Valcovanie2_ServoPracRychl2_MM_s * 100);
			Motion[4].par.acc := (Valcovanie2_ServoPracRychl2_MM_s * 1000);
			Motion[4].par.dec := (Valcovanie2_ServoPracRychl2_MM_s * 1000);
			Motion[4].par.position:= (Valcovanie2_ZadanaPozMM * 100); //180mm

			IF NOT SC_OvlZdvihuRotora.Switch1 THEN
				Motion[4].cmd.moveAbsolute:= TRUE;
				SC_OvlZdvihuRotora.Switch1:= TRUE;
			END_IF

			IF (Valcovanie2_AktualPozMM = Valcovanie2_ZadanaPozMM) AND Motion[4].state.StandStill THEN
				Valcovanie2_ZdvihVPOZICI:= TRUE;
				SC_OvlZdvihuRotora.ResetStep:= TRUE;
				SC_OvlZdvihuRotora.Step:= 0;
			ELSIF Motion[4].status.ActTorque >= 5 THEN
				Motion[4].cmd.halt:= TRUE;
				SC_OvlZdvihuRotora.ResetStep:= TRUE;
				SC_OvlZdvihuRotora.Step:= 0;
			ELSIF diValc2_ZdvihHornyLimit THEN
				Motion[4].cmd.halt:= TRUE;
				Alarmy[56]:= TRUE;
				PoruchaStanicaValcovania2:= TRUE;
			END_IF

	END_CASE

	TaktTime.PT:= T#20s;
	TaktTime();

END_ACTION
```

#### OvlOtacaniaNastroja.st
```iecst
ACTION OvlOtacaniaNastroja:

	//Volanie funkcie SequenceControl//
	SequenceControl(SC:= SC_OvlOtacaniaNastroja);

	CASE SC_OvlOtacaniaNastroja.Step OF

		0:
			SC_OvlOtacaniaNastroja.StepName:= '0 - Nulovanie';
			FM_Menic[3].Input.Command.RunForward:= FALSE;
			FM_Menic[3].Input.Command.RunBackward:= FALSE;
			OtacanieNastroja_VPRED:= FALSE;
			OtacanieNastroja_VZAD:= FALSE;
			TP_Valcovanie2_ZamkniOtacVPRED:= FALSE;
			TP_Valcovanie2_ZamkniOtacVZAD:= FALSE;
			IF SC_Valcovanie2.Step <> 0 THEN
				SC_OvlOtacaniaNastroja.ResetStep:= TRUE;
				SC_OvlOtacaniaNastroja.Step:= 1;
			END_IF

		1:
			SC_OvlOtacaniaNastroja.StepName:= '1 - Rozhodnutie o cinnosti';
			IF OtacanieNastroja_VPRED THEN
				SC_OvlOtacaniaNastroja.Step:= 10;
			ELSIF OtacanieNastroja_VZAD THEN
				SC_OvlOtacaniaNastroja.Step:= 20;
			END_IF

		10:
			SC_OvlOtacaniaNastroja.StepName:= '10 - Otacanie nastroja VPRED';
			SC_OvlOtacaniaNastroja.IdleTime.PT:= T#5s;
			SC_OvlOtacaniaNastroja.AlarmTime.PT:= T#3s;
			FM_Menic[3].Input.HighSpeed:= REAL_TO_INT(Valcovanie2_FM_RychlostOtac_Hz * 10); //v Hz
			FM_Menic[3].Input.AccTime:=  REAL_TO_UINT(Valcovanie2_FM_RozbehRampa_s * 10);  //4s
			FM_Menic[3].Input.DecTime:= REAL_TO_UINT(Valcovanie2_FM_DobehRampa_s * 10);  //4s

			IF NOT SC_OvlOtacaniaNastroja.Switch1 THEN
				FM_Menic[3].Input.Command.RunForward:= TRUE;
				TP_Valcovanie2_ZamkniOtacVZAD:= TRUE;
				SC_OvlOtacaniaNastroja.Switch1:= TRUE;
			END_IF

			IF NOT OtacanieNastroja_VPRED THEN
				FM_Menic[3].Input.Command.RunForward:= FALSE;
			END_IF

			IF NOT OtacanieNastroja_VPRED AND NOT FM_Menic[3].Output.Status.Running THEN
				SC_OvlOtacaniaNastroja.ResetStep:= TRUE;
				SC_OvlOtacaniaNastroja.Step:= 0;
			END_IF

		20:
			SC_OvlOtacaniaNastroja.StepName:= '20 - Otacanie nastroja VZAD';
			SC_OvlOtacaniaNastroja.IdleTime.PT:= T#5s;
			SC_OvlOtacaniaNastroja.AlarmTime.PT:= T#3s;
			FM_Menic[3].Input.HighSpeed:= REAL_TO_INT(Valcovanie2_FM_RychlostOtac_Hz * 10); //v Hz
			FM_Menic[3].Input.AccTime:=  REAL_TO_UINT(Valcovanie2_FM_RozbehRampa_s * 10);  //4s
			FM_Menic[3].Input.DecTime:= REAL_TO_UINT(Valcovanie2_FM_DobehRampa_s * 10);  //4s

			IF NOT SC_OvlOtacaniaNastroja.Switch1 THEN
				FM_Menic[3].Input.Command.RunBackward:= TRUE;
				TP_Valcovanie2_ZamkniOtacVPRED:= TRUE;
				SC_OvlOtacaniaNastroja.Switch1:= TRUE;
			END_IF

			IF NOT OtacanieNastroja_VZAD THEN
				FM_Menic[3].Input.Command.RunBackward:= FALSE;
			END_IF

			IF NOT OtacanieNastroja_VZAD AND NOT FM_Menic[3].Output.Status.Running THEN
				SC_OvlOtacaniaNastroja.ResetStep:= TRUE;
				SC_OvlOtacaniaNastroja.Step:= 0;
			END_IF

	END_CASE

			END_ACTION
```

#### OvlHornehoPritlaku.st
```iecst
ACTION OvlHornehoPritlaku:

	//Volanie funkcie SequenceControl//
	SequenceControl(SC:= SC_OvlHornehoPritlaku);

	CASE SC_OvlHornehoPritlaku.Step OF

		0:
			SC_OvlHornehoPritlaku.StepName:= '0 - Nulovanie';
			HornyPritlak_DOLE:= FALSE;
			HornyPritlak_HORE:= FALSE;
			doValc2_ZdvihPritlakuHORE:= FALSE;
//			doValcovanie2_ZostupPritlakuDOLE:= FALSE;
			IF SC_Valcovanie2.Step <> 0 THEN
				SC_OvlHornehoPritlaku.ResetStep:= TRUE;
				SC_OvlHornehoPritlaku.Step:= 1;
			END_IF

		1:
			SC_OvlHornehoPritlaku.StepName:= '1 - Rozhodnutie o cinnosti';
			IF HornyPritlak_HORE THEN
				SC_OvlHornehoPritlaku.Step:= 10;
			ELSIF HornyPritlak_DOLE THEN
				SC_OvlHornehoPritlaku.Step:= 20;
			END_IF

		10:
			SC_OvlHornehoPritlaku.StepName:= '10 - Zodvihnutie horneho pritlaku hore';
			SC_OvlHornehoPritlaku.IdleTime.PT:= T#3s;
			SC_OvlHornehoPritlaku.AlarmTime.PT:= T#3s;

			IF Valcovanie2_Manual THEN
				SC_OvlHornehoPritlaku.IdleTime.IN:= TRUE;
			ELSE
				SC_OvlHornehoPritlaku.AlarmTime.IN:= TRUE;
			END_IF

			IF NOT SC_OvlHornehoPritlaku.Switch1 THEN
				doValc2_ZostupPritlakuDOLE:= FALSE;
				doValc2_ZdvihPritlakuHORE:= TRUE;
				SC_OvlHornehoPritlaku.Switch1:= TRUE;
			END_IF

			IF SC_OvlHornehoPritlaku.AlarmTime.Q THEN
				Alarmy[57]:= TRUE;
				PoruchaStanicaValcovania2:= TRUE;
			END_IF

			IF diValc2_PritlakZasunuty OR SC_OvlHornehoPritlaku.IdleTime.Q THEN
				SC_OvlHornehoPritlaku.ResetStep:= TRUE;
				SC_OvlHornehoPritlaku.Step:= 0;
			END_IF

		20:
			SC_OvlHornehoPritlaku.StepName:= '20 - Zostup horneho pritlaku dole';
			SC_OvlHornehoPritlaku.IdleTime.PT:= T#3s;
			SC_OvlHornehoPritlaku.AlarmTime.PT:= T#3s;

			IF Valcovanie2_Manual THEN
				SC_OvlHornehoPritlaku.IdleTime.IN:= TRUE;
			ELSE
				SC_OvlHornehoPritlaku.AlarmTime.IN:= TRUE;
			END_IF

			IF NOT SC_OvlHornehoPritlaku.Switch1 THEN
				doValc2_ZdvihPritlakuHORE:= FALSE;
				doValc2_ZostupPritlakuDOLE:= TRUE;
				SC_OvlHornehoPritlaku.Switch1:= TRUE;
			END_IF

			IF SC_OvlHornehoPritlaku.AlarmTime.Q THEN
				Alarmy[58]:= TRUE;
				PoruchaStanicaValcovania2:= TRUE;
			END_IF

			IF diValc2_PritlakVysunuty OR SC_OvlHornehoPritlaku.IdleTime.Q THEN
				SC_OvlHornehoPritlaku.ResetStep:= TRUE;
				SC_OvlHornehoPritlaku.Step:= 0;
			END_IF

	END_CASE

END_ACTION
```

### Program Logical/Program/StanicaMerania (IEC)

#### Main.st - Init, cyclic, exit code
```iecst
PROGRAM _INIT
	(* Insert code here *)

END_PROGRAM

PROGRAM _CYCLIC

	diTlacitko_RotorNG;
	diTlacitko_RotorOK;
	doZelenaLED_Tlacitko_rotor_OK;
	doCervenaLED_Tlacitko_rotor_NG;
	diMeranie_Osciloskop_Stav_NG;
	diMeranie_Osciloskop_Stav_OK;
	doMeranie_Osciloskop_START;
	doMeranie_Osciloskop_STOP;

	//Ovládanie vzorkovacej frekvencie osciloskopu//
	IF RotorOtacaj_VPRED THEN
		doMeranie_Osciloskop_Frekvencia:= Blikac50ms;
	ELSE
		doMeranie_Osciloskop_Frekvencia:= FALSE;
	END_IF

	//Meranie prestoja na stanici merania//
	IF StratovyCas_START THEN
		StratovyCas_Milisekundy:= StratovyCas_Milisekundy + 1;
		IF StratovyCas_Milisekundy >= 1000 THEN
			StratovyCas_Sekundy:= StratovyCas_Sekundy + 1;
			StratovyCas_Milisekundy:= 0;
		END_IF
		IF StratovyCas_Sekundy >= 60 THEN
			StratovyCas_Minuty:= StratovyCas_Minuty + 1;
			StratovyCas_Sekundy:= 0;
		END_IF
		IF StratovyCas_Minuty >= 60 THEN
			StratovyCas_Hodiny:= StratovyCas_Hodiny + 1;
			StratovyCas_Minuty:= 0;
		END_IF
		IF StratovyCas_Hodiny >= 24 THEN
			StratovyCas_RESET:= TRUE;
		END_IF
	END_IF

	IF StratovyCas_RESET THEN
		StratovyCas_Milisekundy:= 0;
		StratovyCas_Sekundy:= 0;
		StratovyCas_Minuty:= 0;
		StratovyCas_Hodiny:= 0;
		StratovyCas_RESET:= FALSE;
	END_IF

	//Volanie podprogramov//
	OvladanieOtacaniaRotora;
	OvladanieZdvihu;

	//Volanie funkcie SequenceControl//
	SequenceControl(SC:= SC_Meranie);

	//Prepočet času merania//
	CasMerania:= REAL_TO_TIME(TP_Meranie_CasMerania*1000);

	//Reset sekcie //
	IF Meranie_Reset OR NOT BezpOkruhOplotenia_Aktivovany OR PoruchaStanicaMerania THEN
		SC_Meranie.Step:= 0;
	END_IF

	CASE SC_Meranie.Step OF

		0:
			SC_Meranie.StepName:='0 - Nulovanie';
			SC_OvlOtacania.Step:= 0;
			SC_OvlZdvihu.Step:= 0;;
			Meranie_Automat:= FALSE;
			Meranie_KoniecVyroby:= FALSE;
			Meranie_KoniecCyklu:= FALSE;
			Meranie_Manual:= FALSE;
			Meranie_PoINIT:= FALSE;
			Meranie_Reset:= FALSE;
			Meranie_UkoncilCyklus:= FALSE;
			Meranie_ObsluhaRozhodla:= FALSE;
			doCervenaLED_Tlacitko_rotor_NG:= FALSE;
			doZelenaLED_Tlacitko_rotor_OK:= FALSE;
			StratovyCas_START:= FALSE;
			doMeranie_Osciloskop_START:= FALSE;
			IF BezpOkruhOplotenia_Aktivovany AND NOT PoruchaStanicaMerania THEN
				SC_Meranie.ResetStep:= TRUE;
				SC_Meranie.Step:= 1;
			END_IF

		1:
			SC_Meranie.StepName:='1 - Rozhodnutie o cinnosti';
			IF Meranie_Automat THEN
				SC_Meranie.Step:= 2;
			ELSIF Meranie_Manual THEN
				SC_Meranie.Step:= 700;
			END_IF

			//********************************************************Inicializácia****************************************************************************//

		2:
			SC_Meranie.StepName:='2 - Inicializacia - cakanie na spustenie';
			SC_Meranie.IdleTime.PT:= T#500ms;
			SC_Meranie.AlarmTime.PT:= T#5s;
			SC_Meranie.IdleTime.IN:= TRUE;

			IF SC_Meranie.IdleTime.Q THEN
				SC_Meranie.ResetStep:= TRUE;
				SC_Meranie.Step:= 3;
			END_IF

		3:
			SC_Meranie.StepName:='2 - Inicializacia - zasunutie zdvihu rotora';
			SC_Meranie.IdleTime.PT:= T#500ms;
			SC_Meranie.AlarmTime.PT:= T#5s;

			IF NOT SC_Meranie.Switch1 THEN
				Rotor_POLOZ:= TRUE;
				SC_Meranie.Switch1:= TRUE;
			END_IF

			IF diMeranie_ZdvihSpodnaPoloha THEN
				RotorOtacaj_VPRED:= TRUE;
				Meranie_PoINIT:= TRUE;
				SC_Meranie.ResetStep:= TRUE;
				SC_Meranie.Step:= 100;
			END_IF

			//********************************************************Automatický režim****************************************************************************//
		100:
			SC_Meranie.StepName:='100 - Automaticky rezim - cakanie na start cyklu';
			SC_Meranie.IdleTime.PT:= T#500ms;
			SC_Meranie.AlarmTime.PT:= T#5s;

           SC_Meranie.IdleTime.IN:= NOT diMeranie_PritomnostRotora;

			IF Meranie_KoniecCyklu THEN
				SC_Meranie.ResetStep:= TRUE;
				SC_Meranie.Step:= 0;
			ELSIF Zariadenie_PrebiehaRevorkRezim THEN
				SC_Meranie.ResetStep:= TRUE;
				SC_Meranie.Step:= 120;
			ELSIF Stol_PoINIT AND NOT Meranie_UkoncilCyklus AND diMeranie_PritomnostRotora AND diStol_SnimacPolohyStola THEN
				Meranie_ObsluhaRozhodla:= FALSE;
				doCervenaLED_Tlacitko_rotor_NG:= FALSE;
				doZelenaLED_Tlacitko_rotor_OK:= FALSE;
				SC_Meranie.ResetStep:= TRUE;
				SC_Meranie.Step:= 101;
			ELSIF Stol_PoINIT AND NOT Meranie_UkoncilCyklus AND NOT diMeranie_PritomnostRotora AND SC_Meranie.IdleTime.Q THEN
				Meranie_ObsluhaRozhodla:= FALSE;
				doCervenaLED_Tlacitko_rotor_NG:= FALSE;
				doZelenaLED_Tlacitko_rotor_OK:= FALSE;
				Stol_Pozicia_1:= 0;
				SC_Meranie.ResetStep:= TRUE;
				SC_Meranie.Step:= 120;
			ELSIF Meranie_KoniecVyroby AND NOT Stol_Automat THEN
				SC_Meranie.ResetStep:= TRUE;
				SC_Meranie.Step:= 0;
			END_IF

		101:
			SC_Meranie.StepName:='101 - Automaticky rezim - zdvih rotora';
			SC_Meranie.IdleTime.PT:= T#1s;
			SC_Meranie.AlarmTime.PT:= T#5s;

			IF NOT SC_Meranie.Switch1 AND SC_OvlZdvihu.Step = 1 THEN
				Rotor_ZDVIHNI:= TRUE;
				SC_Meranie.IdleTime.IN:= TRUE;
				SC_Meranie.Switch1:= TRUE;
			END_IF

			IF diMeranie_ZdvihHornaPoloha THEN
				SC_Meranie.ResetStep:= TRUE;
				SC_Meranie.Step:= 102;
			END_IF

		102:
			SC_Meranie.StepName:='102 - Automaticky rezim - spustenie otacania, cakanie na vysledok merania';
			SC_Meranie.IdleTime.PT:= T#5s;
			SC_Meranie.AlarmTime.PT:= T#2s;
			SC_Meranie.IdleTime.IN:= TRUE;

			IF NOT SC_Meranie.Switch1 THEN
				RotorOtacaj_VPRED:= TRUE;
				doMeranie_Osciloskop_START:= TRUE;
				SC_Meranie.AlarmTime.IN:= TRUE;
				SC_Meranie.Switch1:= TRUE;
			END_IF

			IF SC_Meranie.IdleTime.Q THEN
				StratovyCas_START:= TRUE;
			END_IF

			IF EDGEPOS(diMeranie_Osciloskop_Stav_OK) THEN
				Stol_Pozicia_1:= 1;
				StratovyCas_START:= FALSE;
				doMeranie_Osciloskop_START:= FALSE;
				SC_Meranie.ResetStep:= TRUE;
				SC_Meranie.Step:= 103;
			ELSIF EDGEPOS(diMeranie_Osciloskop_Stav_NG) THEN
				Stol_Pozicia_1:= 2;
				StratovyCas_START:= FALSE;
				doMeranie_Osciloskop_START:= FALSE;
				SC_Meranie.ResetStep:= TRUE;
				SC_Meranie.Step:= 103;
			ELSIF Meranie_KoniecCyklu THEN
				StratovyCas_START:= FALSE;
				doMeranie_Osciloskop_START:= FALSE;
				SC_Meranie.ResetStep:= TRUE;
				SC_Meranie.Step:= 103;
			END_IF

		103:
			SC_Meranie.StepName:='103 - Automaticky rezim - zasunutie zdvihu rotora';
			SC_Meranie.IdleTime.PT:= T#5s;
			SC_Meranie.AlarmTime.PT:= T#5s;

			IF NOT SC_Meranie.Switch1  AND SC_OvlZdvihu.Step = 1 THEN
				Rotor_POLOZ:= TRUE;
				SC_Meranie.Switch1:= TRUE;
			END_IF

			IF diMeranie_ZdvihSpodnaPoloha AND diMeranie_PritomnostRotora AND NOT diMeranie_ZdvihHornaPoloha THEN
				SC_Meranie.ResetStep:= TRUE;
				SC_Meranie.Step:= 120;
			ELSIF diMeranie_ZdvihSpodnaPoloha AND NOT diMeranie_PritomnostRotora THEN
				Alarmy[73]:= TRUE;
				PoruchaStanicaMerania:= TRUE;
			ELSIF diMeranie_ZdvihSpodnaPoloha AND diMeranie_ZdvihHornaPoloha THEN
				Alarmy[73]:= TRUE;
				PoruchaStanicaMerania:= TRUE;
			END_IF

		120:
			SC_Meranie.StepName:='120 - Automaticky rezim - vystavenie signalu ukoncenie pracovneho cyklu';
			SC_Meranie.IdleTime.PT:= T#5s;
			SC_Meranie.AlarmTime.PT:= T#5s;

			Meranie_UkoncilCyklus:= TRUE;
			SC_Meranie.ResetStep:= TRUE;
			SC_Meranie.Step:= 121;

		121:
			SC_Meranie.StepName:='121 - Automaticky rezim - cakanie na otocenie stola';
			SC_Meranie.IdleTime.PT:= T#5s;
			SC_Meranie.AlarmTime.PT:= T#5s;

			IF NOT Meranie_UkoncilCyklus THEN
				SC_Meranie.ResetStep:= TRUE;
				SC_Meranie.Step:= 100;
			ELSIF Meranie_KoniecVyroby AND NOT Stol_Automat THEN
				SC_Meranie.ResetStep:= TRUE;
				SC_Meranie.Step:= 0;
			ELSIF Meranie_KoniecCyklu THEN
				SC_Meranie.ResetStep:= TRUE;
				SC_Meranie.Step:= 0;
			END_IF

			//********************************************************Ručný režim***********************************************************************************//
		700:
			SC_Meranie.StepName:='700 - Rucny rezim';

	END_CASE

				END_PROGRAM

PROGRAM _EXIT
				(* Insert code here *)

				END_PROGRAM
```

#### Variables.var - Local variables
```iecst
VAR
	SC_OvlZdvihu : SequenceControlTyp;
	Rotor_ZDVIHNI : BOOL;
	Rotor_POLOZ : BOOL;
	SC_OvlOtacania : SequenceControlTyp;
	RotorOtacaj_VPRED : BOOL;
	RotorOtacaj_VZAD : BOOL;
	CasMerania : TIME;
END_VAR
```

#### OvladanieZdvihu.st
```iecst
ACTION OvladanieZdvihu:

	//Volanie funkcie SequenceControl//
	SequenceControl(SC:= SC_OvlZdvihu);

	CASE SC_OvlZdvihu.Step OF

		0:
			SC_OvlZdvihu.StepName:= '0 - Nulovanie';
			Rotor_ZDVIHNI:= FALSE;
			Rotor_POLOZ:= FALSE;
			doMeranie_ZDVIH:= FALSE;
			doMeranie_ZOSTUP:= FALSE;
			IF SC_Meranie.Step <> 0 THEN
				SC_OvlZdvihu.ResetStep:= TRUE;
				SC_OvlZdvihu.Step:= 1;
			END_IF

		1:
			SC_OvlZdvihu.StepName:= '1 - Rozhodnutie o cinnosti';
			IF Rotor_ZDVIHNI THEN
				SC_OvlZdvihu.Step:= 10;
			ELSIF Rotor_POLOZ THEN
				SC_OvlZdvihu.Step:= 20;
			END_IF

		10:
			SC_OvlZdvihu.StepName:= '10 - Zodvihnutie rotora';
			SC_OvlZdvihu.IdleTime.PT:= T#1s;
			SC_OvlZdvihu.AlarmTime.PT:= T#3s;
			SC_OvlZdvihu.IdleTime.IN:= TRUE;

			IF NOT SC_OvlZdvihu.Switch1 THEN
				doMeranie_ZDVIH:= TRUE;
				SC_OvlZdvihu.Switch1:= TRUE;
			END_IF

//			IF SC_OvlZdvihu.AlarmTime.Q THEN
//				Alarmy[70]:= TRUE;
//				PoruchaStanicaMerania:= TRUE;
//			END_IF

			IF SC_OvlZdvihu.IdleTime.Q THEN
				SC_OvlZdvihu.ResetStep:= TRUE;
				SC_OvlZdvihu.Step:= 0;
			END_IF

		20:
			SC_OvlZdvihu.StepName:= '20 - Polozenie rotora';
			SC_OvlZdvihu.IdleTime.PT:= T#3s;
			SC_OvlZdvihu.AlarmTime.PT:= T#3s;

			IF Meranie_Manual THEN
				SC_OvlZdvihu.IdleTime.IN:= TRUE;
			ELSE
				SC_OvlZdvihu.AlarmTime.IN:= TRUE;
			END_IF

			IF NOT SC_OvlZdvihu.Switch1 THEN
				doMeranie_ZOSTUP:= TRUE;
				SC_OvlZdvihu.Switch1:= TRUE;
			END_IF

			IF SC_OvlZdvihu.AlarmTime.Q THEN
				Alarmy[71]:= TRUE;
				PoruchaStanicaMerania:= TRUE;
			END_IF

			IF diMeranie_ZdvihSpodnaPoloha OR SC_OvlZdvihu.IdleTime.Q THEN
				SC_OvlZdvihu.ResetStep:= TRUE;
				SC_OvlZdvihu.Step:= 0;
			END_IF

	END_CASE

END_ACTION
```

#### OvladanieOtacaniaRotora.st
```iecst
ACTION OvladanieOtacaniaRotora:

	//Volanie funkcie SequenceControl//
	SequenceControl(SC:= SC_OvlOtacania);

	//Zadanie rýchlosti otáčania rotora//
	Meranie_FM_RychlostOtac_Hz:= TP_Meranie_RychlostOtacania;

	CASE SC_OvlOtacania.Step OF

		0:
			SC_OvlOtacania.StepName:= '0 - Nulovanie';
			FM_Menic[1].Input.Command.RunForward:= FALSE;
			FM_Menic[1].Input.Command.RunBackward:= FALSE;
			RotorOtacaj_VPRED:= FALSE;
			RotorOtacaj_VZAD:= FALSE;
			IF SC_Meranie.Step <> 0 THEN
				SC_OvlOtacania.ResetStep:= TRUE;
				SC_OvlOtacania.Step:= 1;
			END_IF

		1:
			SC_OvlOtacania.StepName:= '1 - Rozhodnutie o cinnosti';
			IF RotorOtacaj_VPRED THEN
				SC_OvlOtacania.Step:= 10;
			ELSIF RotorOtacaj_VZAD THEN
				SC_OvlOtacania.Step:= 20;
			END_IF

		10:
			SC_OvlOtacania.StepName:= '10 - Otacanie rotora VPRED';
			SC_OvlOtacania.IdleTime.PT:= T#5s;
			SC_OvlOtacania.AlarmTime.PT:= T#15s;
			FM_Menic[1].Input.HighSpeed:= (Meranie_FM_RychlostOtac_Hz * 10); //v Hz
			FM_Menic[1].Input.AccTime:= 1;  //0.1s
			FM_Menic[1].Input.DecTime:= 1;  //0.1s
			RotorOtacaj_VZAD:= FALSE;

			IF NOT SC_OvlOtacania.Switch1 THEN
				FM_Menic[1].Input.Command.RunForward:= TRUE;
				SC_OvlOtacania.Switch1:= TRUE;
			END_IF

			IF NOT RotorOtacaj_VPRED THEN
				SC_OvlOtacania.ResetStep:= TRUE;
				SC_OvlOtacania.Step:= 0;
			END_IF

		20:
			SC_OvlOtacania.StepName:= '20 - Otacanie rotora VZAD';
			SC_OvlOtacania.IdleTime.PT:= T#5s;
			SC_OvlOtacania.AlarmTime.PT:= T#15s;
			FM_Menic[1].Input.HighSpeed:= (Meranie_FM_RychlostOtac_Hz * 10); //v Hz
			FM_Menic[1].Input.AccTime:= 1;  //0.1s
			FM_Menic[1].Input.DecTime:= 1;  //0.1s
			RotorOtacaj_VPRED:= FALSE;

			IF NOT SC_OvlOtacania.Switch1 THEN
				FM_Menic[1].Input.Command.RunBackward:= TRUE;
				SC_OvlOtacania.Switch1:= TRUE;
			END_IF

			IF NOT RotorOtacaj_VZAD THEN
				SC_OvlOtacania.ResetStep:= TRUE;
				SC_OvlOtacania.Step:= 0;
			END_IF

	END_CASE

END_ACTION
```

### Program Logical/Program/VystupnyManipulator (IEC)

#### Main.st - Init, cyclic, exit code
```iecst
PROGRAM _INIT
	(* Insert code here *)

END_PROGRAM

PROGRAM _CYCLIC

	//Volanie podprogramov//
	OvladanieGripra;
	OvladaniePojazdu;
	OvladanieZdvihu;

	//Volanie funkcie SequenceControl//
	SequenceControl(SC:= SC_VystupnyManipulator);

	//Reset sekcie //
	IF VystupManipulator_Reset OR NOT BezpOkruhOplotenia_Aktivovany OR PoruchaVystupManipulator THEN
		SC_VystupnyManipulator.Step:= 0;
	END_IF

	CASE SC_VystupnyManipulator.Step OF

		0:
			SC_VystupnyManipulator.StepName:='0 - Nulovanie';
			SC_OvlGripra.Step:= 0;
			SC_OvlServoPojazdu.Step:= 0;
			SC_OvlZdvihu.Step:= 0;
			VystupManipulator_Automat:= FALSE;
			VystupManipulator_KoniecVyroby:= FALSE;
			VystupManipulator_KoniecCyklu:= FALSE;
			VystupManipulator_Manual:= FALSE;
			VystupManipulator_PoINIT:= FALSE;
			VystupManipulator_Reset:= FALSE;
			VystupManipulator_PojazdVPOZICI:= FALSE;
			VystupManipulator_UkoncilCyklus:= FALSE;

			IF BezpOkruhOplotenia_Aktivovany AND NOT PoruchaVystupManipulator THEN
				SC_VystupnyManipulator.ResetStep:= TRUE;
				SC_VystupnyManipulator.Step:= 1;
			END_IF

		1:
			SC_VystupnyManipulator.StepName:='1 - Rozhodnutie o cinnosti';
			IF VystupManipulator_Automat THEN
				SC_VystupnyManipulator.Step:= 2;
			ELSIF VystupManipulator_Manual THEN
				SC_VystupnyManipulator.Step:= 700;
			END_IF

		//********************************************************Inicializácia****************************************************************************//

		2:
			SC_VystupnyManipulator.StepName:='2 - Inicializacia - cakanie na spustenie';
			SC_VystupnyManipulator.IdleTime.PT:= T#500ms;
			SC_VystupnyManipulator.AlarmTime.PT:= T#5s;
			SC_VystupnyManipulator.IdleTime.IN:= TRUE;

			IF SC_VystupnyManipulator.IdleTime.Q THEN
				SC_VystupnyManipulator.ResetStep:= TRUE;
				SC_VystupnyManipulator.Step:= 3;
			END_IF

		3:
			SC_VystupnyManipulator.StepName:='2 - Inicializacia - kontrola home serva';
			SC_VystupnyManipulator.IdleTime.PT:= T#500ms;
			SC_VystupnyManipulator.AlarmTime.PT:= T#5s;

			IF Motion[2].status.DriveStatus.HomingOk THEN
				SC_VystupnyManipulator.ResetStep:= TRUE;
				SC_VystupnyManipulator.Step:= 5;
			ELSE
				SC_VystupnyManipulator.ResetStep:= TRUE;
				SC_VystupnyManipulator.Step:= 4;
			END_IF

		4:
			SC_VystupnyManipulator.StepName:='4 - Inicializacia - homing serva';
			SC_VystupnyManipulator.IdleTime.PT:= T#500ms;
			SC_VystupnyManipulator.AlarmTime.PT:= T#5s;

			IF NOT SC_VystupnyManipulator.Switch1 THEN
				VystupManipulator_PojazdHOME:= TRUE;
				SC_VystupnyManipulator.Switch1:= TRUE;
			END_IF

			IF Motion[2].status.DriveStatus.HomingOk THEN
				SC_VystupnyManipulator.IdleTime.IN:= TRUE;
			END_IF

			IF Motion[2].status.DriveStatus.HomingOk AND SC_VystupnyManipulator.IdleTime.Q AND Motion[2].state.StandStill THEN
				SC_VystupnyManipulator.ResetStep:= TRUE;
				SC_VystupnyManipulator.Step:= 6;
			END_IF

		5:
			SC_VystupnyManipulator.StepName:='5 - Inicializacia - zodvihnutie gripra';
			SC_VystupnyManipulator.IdleTime.PT:= T#500ms;
			SC_VystupnyManipulator.AlarmTime.PT:= T#5s;

			IF NOT SC_VystupnyManipulator.Switch1 THEN
				Zdvih_Manipulatora:= TRUE;
				SC_VystupnyManipulator.Switch1:= TRUE;
			END_IF

			IF diVystupManipul_ZasunutyHore THEN
				SC_VystupnyManipulator.ResetStep:= TRUE;
				SC_VystupnyManipulator.Step:= 6;
			END_IF

		6:
			SC_VystupnyManipulator.StepName:='6 - Inicializacia - rozhodnutie o presunu manipulatora';
			SC_VystupnyManipulator.IdleTime.PT:= T#500ms;
			SC_VystupnyManipulator.AlarmTime.PT:= T#5s;

			IF diVystupManipul_GriperOtvoreny AND diVystupManipul_GriperZatvoreny THEN
				Alarmy[81]:= TRUE;
				PoruchaVystupManipulator:= TRUE;
			ELSIF diVystupManipul_GriperOtvoreny AND NOT diVystupManipul_GriperZatvoreny THEN
				SC_VystupnyManipulator.ResetStep:= TRUE;
				SC_VystupnyManipulator.Step:= 7;
			ELSIF NOT diVystupManipul_GriperOtvoreny AND diVystupManipul_GriperZatvoreny THEN
				SC_VystupnyManipulator.ResetStep:= TRUE;
				SC_VystupnyManipulator.Step:= 8;
			END_IF

		7:
			SC_VystupnyManipulator.StepName:='6 - Inicializacia - presun nad stol';
			SC_VystupnyManipulator.IdleTime.PT:= T#500ms;
			SC_VystupnyManipulator.AlarmTime.PT:= T#5s;

			VystupManipulator_ZadanaPozMM:= TP_VystupManip_PoziciaOdoberania;

			IF NOT SC_VystupnyManipulator.Switch1 THEN
				ServoPojazd_Polohuj:= TRUE;
				SC_VystupnyManipulator.Switch1:= TRUE;
			END_IF

			IF VystupManipulator_PojazdVPOZICI THEN
				VystupManipulator_PojazdVPOZICI:= FALSE;
				VystupManipulator_PoINIT:= TRUE;
				SC_VystupnyManipulator.ResetStep:= TRUE;
				SC_VystupnyManipulator.Step:= 100;
			END_IF

		8:
			SC_VystupnyManipulator.StepName:='8 - Inicializacia - presun nad NG dopravnik';
			SC_VystupnyManipulator.IdleTime.PT:= T#500ms;
			SC_VystupnyManipulator.AlarmTime.PT:= T#5s;

			VystupManipulator_ZadanaPozMM:= TP_VystupManip_PoziciaUklad_NG;

			IF NOT SC_VystupnyManipulator.Switch1 THEN
				ServoPojazd_Polohuj:= TRUE;
				SC_VystupnyManipulator.Switch1:= TRUE;
			END_IF

			IF VystupManipulator_PojazdVPOZICI THEN
				VystupManipulator_PojazdVPOZICI:= FALSE;
				VystupManipulator_PoINIT:= TRUE;
				SC_VystupnyManipulator.ResetStep:= TRUE;
				SC_VystupnyManipulator.Step:= 106;
			END_IF

		//********************************************************Automatický režim****************************************************************************//
		100:
			SC_VystupnyManipulator.StepName:='100 - Automaticky rezim - cakanie na start cyklu';
			SC_VystupnyManipulator.IdleTime.PT:= T#500ms;
			SC_VystupnyManipulator.AlarmTime.PT:= T#5s;

            SC_VystupnyManipulator.IdleTime.IN:= NOT diStol_PritomnostRotoraVystup;

			IF VystupManipulator_KoniecCyklu THEN
				SC_VystupnyManipulator.ResetStep:= TRUE;
				SC_VystupnyManipulator.Step:= 0;
			ELSIF Stol_PoINIT AND NOT VystupManipulator_UkoncilCyklus AND diVystupManipul_GriperOtvoreny AND diStol_PritomnostRotoraVystup AND diStol_SnimacPolohyStola THEN
				SC_VystupnyManipulator.ResetStep:= TRUE;
				SC_VystupnyManipulator.Step:= 102;
			ELSIF Stol_PoINIT AND NOT VystupManipulator_UkoncilCyklus AND NOT diStol_PritomnostRotoraVystup AND SC_VystupnyManipulator.IdleTime.Q THEN
				VystupManipulator_UkoncilCyklus:= TRUE;
				SC_VystupnyManipulator.ResetStep:= TRUE;
				SC_VystupnyManipulator.Step:= 121;
			ELSIF VystupManipulator_KoniecVyroby AND NOT Stol_Automat THEN
				SC_VystupnyManipulator.ResetStep:= TRUE;
				SC_VystupnyManipulator.Step:= 0;
			END_IF

		102:
			SC_VystupnyManipulator.StepName:='102 - Automaticky rezim - zostup gripra';
			SC_VystupnyManipulator.IdleTime.PT:= T#500ms;
			SC_VystupnyManipulator.AlarmTime.PT:= T#5s;

			IF NOT SC_VystupnyManipulator.Switch1 AND SC_OvlZdvihu.Step = 1 THEN
				Zostup_Manipulatora:= TRUE;
				SC_VystupnyManipulator.Switch1:= TRUE;
			END_IF

			IF diVystupManipul_VysunutyDole THEN
				SC_VystupnyManipulator.ResetStep:= TRUE;
				SC_VystupnyManipulator.Step:= 103;
			END_IF

		103:
			SC_VystupnyManipulator.StepName:='103 - Automaticky rezim - zatvorenie gripra';
			SC_VystupnyManipulator.IdleTime.PT:= T#500ms;
			SC_VystupnyManipulator.AlarmTime.PT:= T#5s;

			IF NOT SC_VystupnyManipulator.Switch1 THEN
				Zatvor_Griper:= TRUE;
				SC_VystupnyManipulator.Switch1:= TRUE;
			END_IF

			IF diVystupManipul_GriperZatvoreny THEN
				SC_VystupnyManipulator.ResetStep:= TRUE;
				SC_VystupnyManipulator.Step:= 104;
			END_IF

		104:
			SC_VystupnyManipulator.StepName:='104 - Automaticky rezim - zdvih gripra, vystavenie signalu ukoncenia cyklu';
			SC_VystupnyManipulator.IdleTime.PT:= T#500ms;
			SC_VystupnyManipulator.AlarmTime.PT:= T#5s;
			SC_VystupnyManipulator.IdleTime.IN:= TRUE;

			IF NOT SC_VystupnyManipulator.Switch1 THEN
				Zdvih_Manipulatora:= TRUE;
				SC_VystupnyManipulator.Switch1:= TRUE;
			END_IF

			IF diVystupManipul_ZasunutyHore THEN
				IF Zariadenie_PrebiehaRevorkRezim THEN
					VystupManipulator_Drzi_OK_Kus:= TRUE;
					VystupManipulator_Drzi_NG_Kus:= FALSE;
					VystupManipulator_UkoncilCyklus:= TRUE;
					SC_VystupnyManipulator.ResetStep:= TRUE;
					SC_VystupnyManipulator.Step:= 105;
				ELSIF VystupManipulator_OdoberNGKus THEN
					VystupManipulator_Drzi_NG_Kus:= TRUE;
					VystupManipulator_Drzi_OK_Kus:= FALSE;
					VystupManipulator_OdoberNGKus:= FALSE;
					VystupManipulator_UkoncilCyklus:= TRUE;
					SC_VystupnyManipulator.ResetStep:= TRUE;
					SC_VystupnyManipulator.Step:= 105;
				ELSIF Stol_Pozicia_3 = 2 OR Stol_Pozicia_3 = 0 THEN
					VystupManipulator_Drzi_NG_Kus:= TRUE;
					VystupManipulator_Drzi_OK_Kus:= FALSE;
					VystupManipulator_UkoncilCyklus:= TRUE;
					SC_VystupnyManipulator.ResetStep:= TRUE;
					SC_VystupnyManipulator.Step:= 105;
				ELSIF Stol_Pozicia_3 = 1 THEN
					VystupManipulator_Drzi_OK_Kus:= TRUE;
					VystupManipulator_Drzi_NG_Kus:= FALSE;
					VystupManipulator_UkoncilCyklus:= TRUE;
					SC_VystupnyManipulator.ResetStep:= TRUE;
					SC_VystupnyManipulator.Step:= 105;
				END_IF
			END_IF

		105:
			SC_VystupnyManipulator.StepName:='105 - Automaticky rezim - rozhodnutie o polozeni kusu, presun manipulatora na poziciu ukladania';
			SC_VystupnyManipulator.IdleTime.PT:= T#500ms;
			SC_VystupnyManipulator.AlarmTime.PT:= T#5s;

			IF VystupManipulator_Drzi_NG_Kus THEN
				VystupManipulator_ZadanaPozMM:= TP_VystupManip_PoziciaUklad_NG;  //480;  //Pozícia dopravníka NG
			ELSIF VystupManipulator_Drzi_OK_Kus THEN
				VystupManipulator_ZadanaPozMM:= TP_VystupManip_PoziciaUklad_OK;  //353;  //Pozícia dopravníka OK
			END_IF

			IF NOT SC_VystupnyManipulator.Switch1 THEN
				ServoPojazd_Polohuj:= TRUE;
				SC_VystupnyManipulator.Switch1:= TRUE;
			END_IF

			IF VystupManipulator_PojazdVPOZICI THEN
				VystupManipulator_PojazdVPOZICI:= FALSE;
				SC_VystupnyManipulator.ResetStep:= TRUE;
				SC_VystupnyManipulator.Step:= 106;
			END_IF

		106:
			SC_VystupnyManipulator.StepName:='105 - Automaticky rezim - cakanie na polozenie rotora na dopravnik';
			SC_VystupnyManipulator.IdleTime.PT:= T#500ms;
			SC_VystupnyManipulator.AlarmTime.PT:= T#5s;

			IF (VystupManipulator_AktualPozMM = TP_VystupManip_PoziciaUklad_NG) AND NOT diVystDoprNG_SnimacZaplnTrate AND diVystDopr_OdsuvacZasunuty AND VystupOdsuvac_CakaNaKusy THEN
				SC_VystupnyManipulator.ResetStep:= TRUE;
				SC_VystupnyManipulator.Step:= 107;
			ELSIF (VystupManipulator_AktualPozMM = TP_VystupManip_PoziciaUklad_OK) AND NOT diVystDoprOK_SnimacZaplnTrate AND diVystDopr_OdsuvacZasunuty AND VystupOdsuvac_CakaNaKusy THEN
				SC_VystupnyManipulator.ResetStep:= TRUE;
				SC_VystupnyManipulator.Step:= 107;
			END_IF

		107:
			SC_VystupnyManipulator.StepName:='107 - Automaticky rezim - polozenie rotora na dopravnik';
			SC_VystupnyManipulator.IdleTime.PT:= T#1s;
			SC_VystupnyManipulator.AlarmTime.PT:= T#5s;
			SC_VystupnyManipulator.IdleTime.IN:= TRUE;

			IF NOT SC_VystupnyManipulator.Switch1 THEN
				Zostup_Manipulatora:= TRUE;
				SC_VystupnyManipulator.Switch1:= TRUE;
			END_IF

			IF diVystupManipul_VysunutyDole THEN
				SC_VystupnyManipulator.ResetStep:= TRUE;
				SC_VystupnyManipulator.Step:= 108;
			END_IF

		108:
			SC_VystupnyManipulator.StepName:='108 - Automaticky rezim - otvorenie gripra';
			SC_VystupnyManipulator.IdleTime.PT:= T#500ms;
			SC_VystupnyManipulator.AlarmTime.PT:= T#5s;

			IF NOT SC_VystupnyManipulator.Switch1 THEN
				Otvor_Griper:= TRUE;
				SC_VystupnyManipulator.Switch1:= TRUE;
			END_IF

			IF diVystupManipul_GriperOtvoreny THEN
				VystupManipulator_Drzi_NG_Kus:= FALSE;
				VystupManipulator_Drzi_OK_Kus:= FALSE;
				SC_VystupnyManipulator.ResetStep:= TRUE;
				SC_VystupnyManipulator.Step:= 109;
			END_IF

		109:
			SC_VystupnyManipulator.StepName:='109 - Automaticky rezim - zdvih gripra';
			SC_VystupnyManipulator.IdleTime.PT:= T#500ms;
			SC_VystupnyManipulator.AlarmTime.PT:= T#5s;

			IF NOT SC_VystupnyManipulator.Switch1 THEN
				Zdvih_Manipulatora:= TRUE;
				SC_VystupnyManipulator.Switch1:= TRUE;
			END_IF

			IF diVystupManipul_ZasunutyHore THEN
				VystupOdsuvac_KusyVlozene:= TRUE;
				SC_VystupnyManipulator.ResetStep:= TRUE;
				SC_VystupnyManipulator.Step:= 110;
			END_IF

		110:
			SC_VystupnyManipulator.StepName:='110 - Automaticky rezim - presun do cakacej pozicie nad stol';
			SC_VystupnyManipulator.IdleTime.PT:= T#500ms;
			SC_VystupnyManipulator.AlarmTime.PT:= T#5s;

			VystupManipulator_ZadanaPozMM:= TP_VystupManip_PoziciaOdoberania;

			IF NOT SC_VystupnyManipulator.Switch1 THEN
				ServoPojazd_Polohuj:= TRUE;
				SC_VystupnyManipulator.Switch1:= TRUE;
			END_IF

			IF VystupManipulator_PojazdVPOZICI THEN
				VystupManipulator_PojazdVPOZICI:= FALSE;
				SC_VystupnyManipulator.ResetStep:= TRUE;
				SC_VystupnyManipulator.Step:= 121;
			END_IF

		121:
			SC_VystupnyManipulator.StepName:='121 - Automaticky rezim - cakanie na otocenie stola';
			SC_VystupnyManipulator.IdleTime.PT:= T#500ms;
			SC_VystupnyManipulator.AlarmTime.PT:= T#5s;

			IF NOT VystupManipulator_UkoncilCyklus THEN
				SC_VystupnyManipulator.ResetStep:= TRUE;
				SC_VystupnyManipulator.Step:= 100;
			ELSIF VystupManipulator_KoniecVyroby AND NOT Stol_Automat THEN
				SC_VystupnyManipulator.ResetStep:= TRUE;
				SC_VystupnyManipulator.Step:= 0;
			ELSIF VystupManipulator_KoniecCyklu THEN
				SC_VystupnyManipulator.ResetStep:= TRUE;
				SC_VystupnyManipulator.Step:= 0;
			END_IF

		//********************************************************Ručný režim***********************************************************************************//
		700:
			SC_VystupnyManipulator.StepName:='700 - Rucny rezim';

			//Polohovanie manipulátora//
			IF RR_PoziciaOdoberaniaStol AND SC_OvlServoPojazdu.Step = 1 THEN
				VystupManipul_Rychlost_MM_s:= TP_VystupManip_RychlostPojazdu;
				VystupManipulator_ZadanaPozMM:= TP_VystupManip_PoziciaOdoberania;
				ServoPojazd_Polohuj:= TRUE;
			ELSIF RR_PoziciaUkladaniaNG AND SC_OvlServoPojazdu.Step = 1 THEN
				VystupManipul_Rychlost_MM_s:= TP_VystupManip_RychlostPojazdu;
				VystupManipulator_ZadanaPozMM:= TP_VystupManip_PoziciaUklad_NG;
				ServoPojazd_Polohuj:= TRUE;
			ELSIF RR_PoziciaUkladaniaOK AND SC_OvlServoPojazdu.Step = 1 THEN
				VystupManipul_Rychlost_MM_s:= TP_VystupManip_RychlostPojazdu;
				VystupManipulator_ZadanaPozMM:= TP_VystupManip_PoziciaUklad_OK;
				ServoPojazd_Polohuj:= TRUE;
			END_IF

	END_CASE

				END_PROGRAM

PROGRAM _EXIT
				(* Insert code here *)

				END_PROGRAM
```

#### Variables.var - Local variables
```iecst
VAR
	SC_OvlGripra : SequenceControlTyp;
	Otvor_Griper : BOOL;
	Zatvor_Griper : BOOL;
	SC_OvlZdvihu : SequenceControlTyp;
	Zdvih_Manipulatora : BOOL;
	Zostup_Manipulatora : BOOL;
	SC_OvlServoPojazdu : SequenceControlTyp;
	ServoPojazd_JoggVPRED : BOOL;
	ServoPojazd_JoggVZAD : BOOL;
	ServoPojazd_Polohuj : BOOL;
	KonstantaPojazd_MM : REAL;
	KonstantaPojazd_Servo : REAL;
	RR_PoziciaOdoberaniaStol : BOOL;
	RR_PoziciaUkladaniaNG : BOOL;
	RR_PoziciaUkladaniaOK : BOOL;
END_VAR
```

#### OvladanieGripra.st
```iecst
ACTION OvladanieGripra:

	//Volanie funkcie SequenceControl//
	SequenceControl(SC:= SC_OvlGripra);

	CASE SC_OvlGripra.Step OF

		0:
			SC_OvlGripra.StepName:= '0 - Nulovanie';
			Otvor_Griper:= FALSE;
			Zatvor_Griper:= FALSE;
			doVystupManipul_GriperOTVOR:= FALSE;
			doVystupManipul_GriperZATVOR:= FALSE;
			IF SC_VystupnyManipulator.Step <> 0 THEN
				SC_OvlGripra.ResetStep:= TRUE;
				SC_OvlGripra.Step:= 1;
			END_IF

		1:
			SC_OvlGripra.StepName:= '1 - Rozhodnutie o cinnosti';
			IF Otvor_Griper THEN
				SC_OvlGripra.Step:= 10;
			ELSIF Zatvor_Griper THEN
				SC_OvlGripra.Step:= 20;
			END_IF

		10:
			SC_OvlGripra.StepName:= '10 - Otvorenie gripra';
			SC_OvlGripra.IdleTime.PT:= T#3s;
			SC_OvlGripra.AlarmTime.PT:= T#3s;

			IF VystupManipulator_Manual THEN
				SC_OvlGripra.IdleTime.IN:= TRUE;
			ELSE
				SC_OvlGripra.AlarmTime.IN:= TRUE;
			END_IF

			IF NOT SC_OvlGripra.Switch1 THEN
				doVystupManipul_GriperOTVOR:= TRUE;
				SC_OvlGripra.Switch1:= TRUE;
			END_IF

			IF SC_OvlGripra.AlarmTime.Q THEN
				Alarmy[81]:= TRUE;
				PoruchaVystupManipulator:= TRUE;
			END_IF

			IF diVystupManipul_GriperOtvoreny OR SC_OvlGripra.IdleTime.Q THEN
				SC_OvlGripra.ResetStep:= TRUE;
				SC_OvlGripra.Step:= 0;
			END_IF

		20:
			SC_OvlGripra.StepName:= '20 - Zatvorenie gripra';
			SC_OvlGripra.IdleTime.PT:= T#3s;
			SC_OvlGripra.AlarmTime.PT:= T#3s;

			IF VystupManipulator_Manual THEN
				SC_OvlGripra.IdleTime.IN:= TRUE;
			ELSE
				SC_OvlGripra.AlarmTime.IN:= TRUE;
			END_IF

			IF NOT SC_OvlGripra.Switch1 THEN
				doVystupManipul_GriperZATVOR:= TRUE;
				SC_OvlGripra.Switch1:= TRUE;
			END_IF

			IF SC_OvlGripra.AlarmTime.Q THEN
				Alarmy[80]:= TRUE;
				PoruchaVystupManipulator:= TRUE;
			END_IF

			IF diVystupManipul_GriperZatvoreny OR SC_OvlGripra.IdleTime.Q THEN
				SC_OvlGripra.ResetStep:= TRUE;
				SC_OvlGripra.Step:= 0;
			END_IF

	END_CASE

END_ACTION
```

#### OvladanieZdvihu.st
```iecst
ACTION OvladanieZdvihu:

	//Volanie funkcie SequenceControl//
	SequenceControl(SC:= SC_OvlZdvihu);

	CASE SC_OvlZdvihu.Step OF

		0:
			SC_OvlZdvihu.StepName:= '0 - Nulovanie';
			Zdvih_Manipulatora:= FALSE;
			Zostup_Manipulatora:= FALSE;
			doVystupManipul_ZDVIH:= FALSE;
			doVystupManipul_ZOSTUP:= FALSE;
			IF SC_VystupnyManipulator.Step <> 0 THEN
				SC_OvlZdvihu.ResetStep:= TRUE;
				SC_OvlZdvihu.Step:= 1;
			END_IF

		1:
			SC_OvlZdvihu.StepName:= '1 - Rozhodnutie o cinnosti';
			IF Zdvih_Manipulatora THEN
				SC_OvlZdvihu.Step:= 10;
			ELSIF Zostup_Manipulatora THEN
				SC_OvlZdvihu.Step:= 20;
			END_IF

		10:
			SC_OvlZdvihu.StepName:= '10 - Zdvih manipulatora';
			SC_OvlZdvihu.IdleTime.PT:= T#3s;
			SC_OvlZdvihu.AlarmTime.PT:= T#3s;

			IF VystupManipulator_Manual THEN
				SC_OvlZdvihu.IdleTime.IN:= TRUE;
			ELSE
				SC_OvlZdvihu.AlarmTime.IN:= TRUE;
			END_IF

			IF NOT SC_OvlZdvihu.Switch1 THEN
				doVystupManipul_ZDVIH:= TRUE;
				SC_OvlZdvihu.Switch1:= TRUE;
			END_IF

			IF SC_OvlZdvihu.AlarmTime.Q THEN
				Alarmy[82]:= TRUE;
				PoruchaVystupManipulator:= TRUE;
			END_IF

			IF diVystupManipul_ZasunutyHore OR SC_OvlZdvihu.IdleTime.Q THEN
				SC_OvlZdvihu.ResetStep:= TRUE;
				SC_OvlZdvihu.Step:= 0;
			END_IF

		20:
			SC_OvlZdvihu.StepName:= '20 - Zostup manipulatora';
			SC_OvlZdvihu.IdleTime.PT:= T#1s;
			SC_OvlZdvihu.AlarmTime.PT:= T#3s;
			SC_OvlZdvihu.IdleTime.IN:= TRUE;

			IF NOT SC_OvlZdvihu.Switch1 THEN
				doVystupManipul_ZOSTUP:= TRUE;
				SC_OvlZdvihu.Switch1:= TRUE;
			END_IF

			IF EDGEPOS (diVystupManipul_ZdvihStredPoloha = TRUE) THEN
				doVystupManipul_ZDVIH:= TRUE;
			END_IF

			IF diVystupManipul_VysunutyDole OR SC_OvlZdvihu.IdleTime.Q THEN
				SC_OvlZdvihu.ResetStep:= TRUE;
				SC_OvlZdvihu.Step:= 0;
			END_IF

	END_CASE

END_ACTION
```

#### OvladaniePojazdu.st
```iecst
ACTION OvladaniePojazdu:

	//Prepočet rýchlosti pojazdu manipulátora//
	KonstantaPojazd_MM:= 8;  //8mm
	KonstantaPojazd_Servo:= 800; //počet jednotiek za 8mm

	VystupManipul_Rychlost_MM_s:= TP_VystupManip_RychlostPojazdu;
	VystupManipulator_RychlostPoloho:= (VystupManipul_Rychlost_MM_s / KonstantaPojazd_MM) * KonstantaPojazd_Servo;
	VystupManipulator_RychlJoggingu:= (VystupManipul_RychlostJog_MM_s / KonstantaPojazd_MM) * KonstantaPojazd_Servo;
	VystupManipulator_AktualPozMM;

	//Volanie funkcie SequenceControl//
	SequenceControl(SC:= SC_OvlServoPojazdu);

	CASE SC_OvlServoPojazdu.Step OF

		0:
			SC_OvlServoPojazdu.StepName:= '0 - Nulovanie';
			ServoPojazd_JoggVPRED:= FALSE;
			ServoPojazd_JoggVZAD:= FALSE;
			ServoPojazd_Polohuj:= FALSE;
			VystupManipulator_PojazdHOME:= FALSE;
			Motion[2].cmd.home:= FALSE;
			Motion[2].cmd.moveAbsolute:= FALSE;
			Motion[2].cmd.moveJogNeg:= FALSE;
			Motion[2].cmd.moveJogPos:= FALSE;
			VystupManipulator_PrebiehaHoming:= FALSE;
			IF NOT SC_OvlServoPojazdu.Switch1 AND Motion[2].status.DriveStatus.HomingOk THEN
				Motion[2].cmd.halt:= TRUE;
				SC_OvlServoPojazdu.Switch1:= TRUE;
			END_IF
			IF SC_VystupnyManipulator.Step <> 0 THEN
				SC_OvlServoPojazdu.ResetStep:= TRUE;
				SC_OvlServoPojazdu.Step:= 1;
			END_IF

		1:
			SC_OvlServoPojazdu.StepName:= '1 - Rozhodnutie o cinnosti';
			IF ServoPojazd_JoggVPRED THEN
				SC_OvlServoPojazdu.Step:= 10;
			ELSIF ServoPojazd_JoggVZAD THEN
				SC_OvlServoPojazdu.Step:= 20;
			ELSIF ServoPojazd_Polohuj THEN
				SC_OvlServoPojazdu.Step:= 30;
			ELSIF VystupManipulator_PojazdHOME THEN
				SC_OvlServoPojazdu.Step:= 40;
			END_IF

		10:
			SC_OvlServoPojazdu.StepName:= '10 - Jogging VPRED';
			SC_OvlServoPojazdu.IdleTime.PT:= T#3s;
			SC_OvlServoPojazdu.AlarmTime.PT:= T#3s;

			Motion[2].par.velocityJog:= VystupManipulator_RychlJoggingu;
			Motion[2].par.acc := (VystupManipulator_RychlJoggingu*10);
			Motion[2].par.dec := (VystupManipulator_RychlJoggingu*10);

			IF NOT SC_OvlServoPojazdu.Switch1 THEN
				Motion[2].cmd.moveJogPos:= TRUE;
				SC_OvlServoPojazdu.Switch1:= TRUE;
			END_IF

			IF NOT ServoPojazd_JoggVPRED OR diVystupManipul_PrednyLimSnimac OR VystupManipulator_AktualPozMM >= 360 OR NOT diVystupManipul_ZasunutyHore THEN
				SC_OvlServoPojazdu.ResetStep:= TRUE;
				SC_OvlServoPojazdu.Step:= 0;
			END_IF

		20:
			SC_OvlServoPojazdu.StepName:= '10 - Jogging VZAD';
			SC_OvlServoPojazdu.IdleTime.PT:= T#3s;
			SC_OvlServoPojazdu.AlarmTime.PT:= T#3s;

			Motion[2].par.velocityJog:= VystupManipulator_RychlJoggingu;
			Motion[2].par.acc := (VystupManipulator_RychlJoggingu*10);
			Motion[2].par.dec := (VystupManipulator_RychlJoggingu*10);

			IF NOT SC_OvlServoPojazdu.Switch1 THEN
				Motion[2].cmd.moveJogNeg:= TRUE;
				SC_OvlServoPojazdu.Switch1:= TRUE;
			END_IF

			IF NOT ServoPojazd_JoggVZAD OR diVystupManipul_ZadnyLimSnimac OR VystupManipulator_AktualPozMM <= 0 OR NOT diVystupManipul_ZasunutyHore THEN
				SC_OvlServoPojazdu.ResetStep:= TRUE;
				SC_OvlServoPojazdu.Step:= 0;
			END_IF

		30:
			SC_OvlServoPojazdu.StepName:= '30 - Start polohovanie pojazdu';
			SC_OvlServoPojazdu.IdleTime.PT:= T#3s;
			SC_OvlServoPojazdu.AlarmTime.PT:= T#3s;

			Motion[2].par.velocity:= VystupManipulator_RychlostPoloho;
			Motion[2].par.acc := (VystupManipulator_RychlostPoloho*10);
			Motion[2].par.dec := (VystupManipulator_RychlostPoloho*10);
			Motion[2].par.position:= (VystupManipulator_ZadanaPozMM * 100);

			IF NOT SC_OvlServoPojazdu.Switch1 THEN
				Motion[2].cmd.moveAbsolute:= TRUE;
				SC_OvlServoPojazdu.Switch1:= TRUE;
			END_IF

			IF NOT Motion[2].state.StandStill THEN
				SC_OvlServoPojazdu.ResetStep:= TRUE;
				SC_OvlServoPojazdu.Step:= 31;
			ELSIF (VystupManipulator_AktualPozMM = VystupManipulator_ZadanaPozMM) THEN
				SC_OvlServoPojazdu.ResetStep:= TRUE;
				SC_OvlServoPojazdu.Step:= 31;
			END_IF

		31:

			SC_OvlServoPojazdu.StepName:= '31 - Ukoncenie polohovanie pojazdu';
			SC_OvlServoPojazdu.IdleTime.PT:= T#3s;
			SC_OvlServoPojazdu.AlarmTime.PT:= T#3s;

			IF Motion[2].state.StandStill (*AND (VystupManipulator_AktualPozMM = VystupManipulator_ZadanaPozMM)*) THEN
				VystupManipulator_PojazdVPOZICI:= TRUE;
				SC_OvlServoPojazdu.ResetStep:= TRUE;
				SC_OvlServoPojazdu.Step:= 0;
			END_IF

			IF diVystupManipul_PrednyLimSnimac OR diVystupManipul_ZadnyLimSnimac THEN
				Alarmy[86]:= TRUE;
				PoruchaVystupManipulator:= TRUE;
			END_IF

		40:
			SC_OvlServoPojazdu.StepName:= '40 - Homing,zdvihnutie gripra';
			SC_OvlServoPojazdu.IdleTime.PT:= T#3s;
			SC_OvlServoPojazdu.AlarmTime.PT:= T#3s;

			IF NOT SC_OvlServoPojazdu.Switch1 THEN
				Zdvih_Manipulatora:= TRUE;
				SC_OvlServoPojazdu.Switch1:= TRUE;
			END_IF

			IF diVystupManipul_ZasunutyHore THEN
				SC_OvlServoPojazdu.ResetStep:= TRUE;
				SC_OvlServoPojazdu.Step:= 41;
			END_IF

		41:
			SC_OvlServoPojazdu.StepName:= '41 - Homing,spustenie';
			SC_OvlServoPojazdu.IdleTime.PT:= T#3s;
			SC_OvlServoPojazdu.AlarmTime.PT:= T#3s;

			IF NOT SC_OvlServoPojazdu.Switch1 THEN
				Motion[2].cmd.home:= TRUE;
				VystupManipulator_PrebiehaHoming:= TRUE;
				SC_OvlServoPojazdu.Switch1:= TRUE;
			END_IF

			IF Motion[2].state.Homing THEN
				SC_OvlServoPojazdu.ResetStep:= TRUE;
				SC_OvlServoPojazdu.Step:= 42;
			END_IF

		42:
			SC_OvlServoPojazdu.StepName:= '42 - Homing,ukoncenie';
			SC_OvlServoPojazdu.IdleTime.PT:= T#3s;
			SC_OvlServoPojazdu.AlarmTime.PT:= T#3s;

			IF Motion[2].status.DriveStatus.HomingOk THEN
				SC_OvlServoPojazdu.ResetStep:= TRUE;
				SC_OvlServoPojazdu.Step:= 0;
			END_IF

	END_CASE

END_ACTION
```

### Program Logical/Program/VystupnyOdsuvac (IEC)

#### Main.st - Init, cyclic, exit code
```iecst
PROGRAM _INIT
	(* Insert code here *)

END_PROGRAM

PROGRAM _CYCLIC

	//Volanie podprogramov//
	OvladanieOdsuvania;

	//Volanie funkcie SequenceControl//
	SequenceControl(SC:= SC_VystupnyOdsuvac);

	//Reset sekcie //
	IF VystupOdsuvac_Reset OR NOT BezpOkruhOplotenia_Aktivovany OR PoruchaVystupOdsuvac THEN
		SC_VystupnyOdsuvac.Step:= 0;
	END_IF

	CASE SC_VystupnyOdsuvac.Step OF

		0:
			SC_VystupnyOdsuvac.StepName:='0 - Nulovanie';
			SC_OvlOdsuvaca.Step:= 0;
			VystupOdsuvac_Automat:= FALSE;
			VystupOdsuvac_KoniecVyroby:= FALSE;
			VystupOdsuvac_KoniecCyklu:= FALSE;
			VystupOdsuvac_Manual:= FALSE;
			VystupOdsuvac_PoINIT:= FALSE;
			VystupOdsuvac_Reset:= FALSE;
			VystupOdsuvac_CakaNaKusy:= FALSE;
			VystupOdsuvac_KusyVlozene:= FALSE;
			IF BezpOkruhOplotenia_Aktivovany AND NOT PoruchaVystupOdsuvac THEN
				SC_VystupnyOdsuvac.ResetStep:= TRUE;
				SC_VystupnyOdsuvac.Step:= 1;
			END_IF

		1:
			SC_VystupnyOdsuvac.StepName:='1 - Rozhodnutie o cinnosti';
			IF VystupOdsuvac_Automat THEN
				SC_VystupnyOdsuvac.Step:= 2;
			ELSIF VystupOdsuvac_Manual THEN
				SC_VystupnyOdsuvac.Step:= 700;
			END_IF

		//********************************************************Inicializácia****************************************************************************//

		2:
			SC_VystupnyOdsuvac.StepName:='2 - Inicializacia - cakanie na spustenie';
			SC_VystupnyOdsuvac.IdleTime.PT:= T#500ms;
			SC_VystupnyOdsuvac.AlarmTime.PT:= T#5s;
			SC_VystupnyOdsuvac.IdleTime.IN:= TRUE;

			IF SC_VystupnyOdsuvac.IdleTime.Q THEN
				SC_VystupnyOdsuvac.ResetStep:= TRUE;
				SC_VystupnyOdsuvac.Step:= 3;
			END_IF

		3:
			SC_VystupnyOdsuvac.StepName:='3 - Inicializacia - vysunutie odsuvaca vpred';
			SC_VystupnyOdsuvac.IdleTime.PT:= T#500ms;
			SC_VystupnyOdsuvac.AlarmTime.PT:= T#5s;

			IF NOT SC_VystupnyOdsuvac.Switch1 AND NOT diVystDoprNG_SnimacZaplnTrate AND NOT diVystDoprOK_SnimacZaplnTrate THEN
				Odsuvac_VYSUN:= TRUE;
				SC_VystupnyOdsuvac.Switch1:= TRUE;
			END_IF

			IF diVystDopr_OdsuvacVysunuty THEN
				SC_VystupnyOdsuvac.ResetStep:= TRUE;
				SC_VystupnyOdsuvac.Step:= 4;
			END_IF

		4:
			SC_VystupnyOdsuvac.StepName:='4 - Inicializacia - zasunutie odsuvaca vzad';
			SC_VystupnyOdsuvac.IdleTime.PT:= T#500ms;
			SC_VystupnyOdsuvac.AlarmTime.PT:= T#5s;

			IF NOT SC_VystupnyOdsuvac.Switch1 AND SC_OvlOdsuvaca.Step = 1 THEN
				Odsuvac_ZASUN:= TRUE;
				SC_VystupnyOdsuvac.Switch1:= TRUE;
			END_IF

			IF diVystDopr_OdsuvacZasunuty THEN
				VystupOdsuvac_PoINIT:= TRUE;
				SC_VystupnyOdsuvac.ResetStep:= TRUE;
				SC_VystupnyOdsuvac.Step:= 100;
			END_IF

		//********************************************************Automatický režim****************************************************************************//
		100:
			SC_VystupnyOdsuvac.StepName:='100 - Automaticky rezim - cakanie na vysunutie';
			SC_VystupnyOdsuvac.IdleTime.PT:= T#500ms;
			SC_VystupnyOdsuvac.AlarmTime.PT:= T#5s;

			IF NOT SC_VystupnyOdsuvac.Switch1 THEN
				VystupOdsuvac_CakaNaKusy:= TRUE;
				SC_VystupnyOdsuvac.Switch1:= TRUE;
			END_IF

			IF VystupOdsuvac_KusyVlozene THEN
				VystupOdsuvac_CakaNaKusy:= FALSE;
				VystupOdsuvac_KusyVlozene:= FALSE;
				SC_VystupnyOdsuvac.ResetStep:= TRUE;
				SC_VystupnyOdsuvac.Step:= 101;
			ELSIF VystupOdsuvac_KoniecVyroby AND NOT VystupManipulator_Automat THEN
				SC_VystupnyOdsuvac.ResetStep:= TRUE;
				SC_VystupnyOdsuvac.Step:= 0;
			ELSIF VystupOdsuvac_KoniecCyklu AND NOT VystupManipulator_Automat THEN
				SC_VystupnyOdsuvac.ResetStep:= TRUE;
				SC_VystupnyOdsuvac.Step:= 0;
			END_IF

		101:
			SC_VystupnyOdsuvac.StepName:='101 - Automaticky rezim - vysunutie odsuvaca vpred';
			SC_VystupnyOdsuvac.IdleTime.PT:= T#500ms;
			SC_VystupnyOdsuvac.AlarmTime.PT:= T#5s;

			IF NOT SC_VystupnyOdsuvac.Switch1 AND NOT diVystDoprNG_SnimacZaplnTrate AND NOT diVystDoprOK_SnimacZaplnTrate THEN
				Odsuvac_VYSUN:= TRUE;
				SC_VystupnyOdsuvac.Switch1:= TRUE;
			END_IF

			IF diVystDopr_OdsuvacVysunuty THEN
				SC_VystupnyOdsuvac.ResetStep:= TRUE;
				SC_VystupnyOdsuvac.Step:= 102;
			END_IF

		102:
			SC_VystupnyOdsuvac.StepName:='101 - Automaticky rezim - zasunutie odsuvaca vzad';
			SC_VystupnyOdsuvac.IdleTime.PT:= T#500ms;
			SC_VystupnyOdsuvac.AlarmTime.PT:= T#5s;

			IF NOT SC_VystupnyOdsuvac.Switch1 AND SC_OvlOdsuvaca.Step = 1 THEN
				Odsuvac_ZASUN:= TRUE;
				SC_VystupnyOdsuvac.Switch1:= TRUE;
			END_IF

			IF diVystDopr_OdsuvacZasunuty THEN
				SC_VystupnyOdsuvac.ResetStep:= TRUE;
				SC_VystupnyOdsuvac.Step:= 100;
			END_IF

		//********************************************************Ručný režim***********************************************************************************//
		700:
			SC_VystupnyOdsuvac.StepName:='700 - Rucny rezim';

	END_CASE

				END_PROGRAM

PROGRAM _EXIT
				(* Insert code here *)

				END_PROGRAM
```

#### Variables.var - Local variables
```iecst
VAR
	SC_OvlOdsuvaca : SequenceControlTyp;
	Odsuvac_VYSUN : BOOL;
	Odsuvac_ZASUN : BOOL;
END_VAR
```

#### OvladanieOdsuvania.st
```iecst
ACTION OvladanieOdsuvania:

	//Volanie funkcie SequenceControl//
	SequenceControl(SC:= SC_OvlOdsuvaca);

	CASE SC_OvlOdsuvaca.Step OF

		0:
			SC_OvlOdsuvaca.StepName:= '0 - Nulovanie';
			Odsuvac_VYSUN:= FALSE;
			Odsuvac_ZASUN:= FALSE;
			doVystDopr_OdsuvacZASUN:= FALSE;
			doVystDopr_OdsuvacVYSUN:= FALSE;
			IF SC_VystupnyOdsuvac.Step <> 0 THEN
				SC_OvlOdsuvaca.ResetStep:= TRUE;
				SC_OvlOdsuvaca.Step:= 1;
			END_IF

		1:
			SC_OvlOdsuvaca.StepName:= '1 - Rozhodnutie o cinnosti';
			IF Odsuvac_VYSUN THEN
				SC_OvlOdsuvaca.Step:= 10;
			ELSIF Odsuvac_ZASUN THEN
				SC_OvlOdsuvaca.Step:= 20;
			END_IF

		10:
			SC_OvlOdsuvaca.StepName:= '10 - Vysunutie odsuvaca vpred';
			SC_OvlOdsuvaca.IdleTime.PT:= T#3s;
			SC_OvlOdsuvaca.AlarmTime.PT:= T#3s;

			IF VystupOdsuvac_Manual THEN
				SC_OvlOdsuvaca.IdleTime.IN:= TRUE;
			ELSE
				SC_OvlOdsuvaca.AlarmTime.IN:= TRUE;
			END_IF

			IF NOT SC_OvlOdsuvaca.Switch1 THEN
				doVystDopr_OdsuvacVYSUN:= TRUE;
				SC_OvlOdsuvaca.Switch1:= TRUE;
			END_IF

			IF SC_OvlOdsuvaca.AlarmTime.Q THEN
				Alarmy[90]:= TRUE;
				PoruchaVystupOdsuvac:= TRUE;
			END_IF

			IF diVystDopr_OdsuvacVysunuty OR SC_OvlOdsuvaca.IdleTime.Q THEN
				SC_OvlOdsuvaca.ResetStep:= TRUE;
				SC_OvlOdsuvaca.Step:= 0;
			END_IF

		20:
			SC_OvlOdsuvaca.StepName:= '20 - Zasunutie odsuvaca vzad';
			SC_OvlOdsuvaca.IdleTime.PT:= T#3s;
			SC_OvlOdsuvaca.AlarmTime.PT:= T#3s;

			IF VystupOdsuvac_Manual THEN
				SC_OvlOdsuvaca.IdleTime.IN:= TRUE;
			ELSE
				SC_OvlOdsuvaca.AlarmTime.IN:= TRUE;
			END_IF

			IF NOT SC_OvlOdsuvaca.Switch1 THEN
				doVystDopr_OdsuvacZASUN:= TRUE;
				SC_OvlOdsuvaca.Switch1:= TRUE;
			END_IF

			IF SC_OvlOdsuvaca.AlarmTime.Q THEN
				Alarmy[91]:= TRUE;
				PoruchaVystupOdsuvac:= TRUE;
			END_IF

			IF diVystDopr_OdsuvacZasunuty OR SC_OvlOdsuvaca.IdleTime.Q THEN
				SC_OvlOdsuvaca.ResetStep:= TRUE;
				SC_OvlOdsuvaca.Step:= 0;
			END_IF

	END_CASE

END_ACTION
```

### Program Logical/Program/Poruchy_Signalizacie (IEC)

#### Main.st - Init, cyclic, exit code
```iecst
PROGRAM _INIT
	(* Insert code here *)

END_PROGRAM

PROGRAM _CYCLIC
	//0 - Porucha tlaku vzduchu//
	//1 - Bolo stlacene tlacitko CS//
	//2 - Hydraulicke cerpadlo - nizka hladina oleja//
	//3 - Hydraulicke cerpadlo - porucha motora cerpadla//
	//4 - Hydraulicke cerpadlo - vysoka teplota oleja//
	//5 - Hydraulicke cerpadlo - zanesenie olejoveho filtra//
	//10 - Oddelovac - porucha prepnutia oddelovaca //
	//15 - Vstupny dopravnik - porucha vysunutia zdvihu rotora//
	//16 - Vstupny dopravnik - porucha zasunutia zdvihu rotora//
	//17 - Vstupny dopravnik - porucha zdvihu rotora//
	//20 - Vstupny manipulator - porucha zatvorenia gripra//
	//21 - Vstupny manipulator - porucha otvorenia gripra//
	//22 - Vstupny manipulátor - porucha zdvihu//
	//23 - Vstupny manipulator - porucha zostupu//
	//24 - Vstupny manipulator - porucha serva pojazdu//
	//25 - Vstupny manipulator - pretazenie serva pojazdu//
	//26 - Vstupny manipulator - dosiahnuta limitna pozicia pojazdu//
	//30 - Otocny stol - porucha motora//
	//31 - Otocny stol - porucha otocenia stola//
	//32 - Otocny stol - vysoka teplota motora//
	//33 - Otocny stol - blokacia stola aktivna//
    //34 - Otocny stol - naliatok nebol odstrihnuty //
	//40 - Stanica strihania - porucha zdvihu rotora//
	//41 - Stanica strihania - porucha zostupu rotora//
	//42 - Stanica strihania - porucha otvorenia gripra naliatku//
	//43 - Stanica strihania - porucha zatvorenia gripra naliatku//
	//44 - Stanica strihania - porucha otvorenia gripra striznika//
	//45 - Stanica strihania - porucha zatvorenia gripra striznika//
	//46 - Stanica strihania - porucha presunu griprov do vychodiskovej pozicie//
	//47 - Stanica strihania - porucha presunu griprov do pozicie odhodenia//
	//48 - Stanica strihania - v stanici zostal zaseknuty rotor//
	//50 - Stanica razenia - porucha zdvihu rotora//
	//51 - Stanica razenia - porucha zostupu rotora//
	//52 - Stanica razenia - v stanici zostal zaseknuty rotor//
	//53 - Stanica vonkajsieho valcovania - porucha serva zdvihu rotora//
	//54 - Stanica vonkajsieho valcovania - porucha menica otacania nastroja//
	//55 - Stanica vonkajsieho valcovania - pretazenie serva zdvihu rotora//
	//56 - Stanica vonkajsieho valcovania - dosiahnuta limitna pozicia zdvihu rotora//
	//57 - Stanica vonkajsieho valcovania - porucha zdvihu horneho pritlaku//
	//58 - Stanica vonkajsieho valcovania - porucha zostupu horneho pritlaku//
	//59 - Stanica vonkajsieho valcovania - nizky tlak vzduchu v hornom pritlaku//
	//60 - Stanica vnutorneho valcovania - porucha zdvihu rotora//
	//61 - Stanica vnutorneho valcovania - porucha zostupu rotora//
	//62 - Stanica vnutorneho valcovania - zatvorenia gripra//
	//63 - Stanica vnutorneho valcovania - otvorenie gripra//
	//64 - Stanica vnutorneho valcovania - porucha motora otacania rotora//
	//65 - Stanica vnutorneho valcovania - porucha serva zdvihu//
	//66 - Stanica vnutorneho valcovania - pretazenie serva zdvihu//
	//67 - Stanica vnutorneho valcovania - dosiahnuta limitna pozicia zdvihu//
	//68 - Stanica vnutorneho valcovania - vypadnuty nastroj valcovania//
	//70 - Stanica merania - porucha zdvihu rotora//
	//71 - Stanica merania - porucha zostupu rotora//
	//72 - Stanica merania - porucha motora otacania rotora//
	//73 - Stanica merania - v stanici zostal zaseknuty rotor//
	//74 - Stanica vonkajsieho valcovania - v stanici zostal zaseknuty rotor//
	//75 - Stanica vonkajsieho valcovania - rotor nebol vyvalcovany//
	//76 - Stanica vonkajsieho valcovania - porucha otáčania valcovacieho nastroja//
	//80 - Vystupny manipulator - porucha zatvorenia gripra//
	//81 - Vystupny manipulator - porucha otvorenia gripra//
	//82 - Vystupny manipulator - porucha zdvihu//
	//83 - Vystupny manipulator - porucha zostupu//
	//84 - Vystupny manipulator - porucha serva pojazdu//
	//85 - Vystupny manipulator - pretazenie serva pojazdu//
	//86 - Vystupny manipulator - dosiahnuta limitna pozicia pojazdu//
	//90 - Vystupny odsuvac - porucha vysunutia//
	//91 - Vystupny odsuvac - porucha zasunutia//
	//92 - Porucha modulu DB1//
	//93 - Porucha modulu DB2//
	//94 - Porucha modulu DB3//
	//95 - Porucha modulu DB4//
	//96 - Porucha modulu DB5//
	//97 - Porucha modulu DB6//

	//*********************************Zistenie alarmu************************************************************//
	FOR i:=0 TO 100 BY 1 DO
		Alarmy[i];
		IF Alarmy[i] = TRUE THEN
			NastalaPorucha:= TRUE;
		END_IF
	END_FOR

	//*********************************Blikanie symbolu poruchy na OP*****************************************//
	IF NastalaPorucha THEN
		ZobrazSymbolAlarmu:= Blikac500ms;
	ELSE
		ZobrazSymbolAlarmu:= FALSE;
	END_IF

	//*********************************Ovládanie kontrolky poruchy********************************************//
	IF NastalaPorucha THEN
		doKontrolkaPORUCHA:= Blikac500ms;
	ELSE
		doKontrolkaPORUCHA:= FALSE;
	END_IF

	//*********************************Zelené svetlo majáka****************************************************//
	IF Zariadenie_StavAutomat AND NOT Zariadenie_StavPoINIT THEN
		doMajak_ZeleneSvetlo:= Blikac500ms;
	ELSIF Zariadenie_StavAutomat AND Zariadenie_StavPoINIT THEN
		doMajak_ZeleneSvetlo:= TRUE;
	ELSE
		doMajak_ZeleneSvetlo:= FALSE;
	END_IF

	//**********************************Žlté svetlo majáka*****************************************************//
	IF TP_ZobrazHlasenieDoprOK_Plny = 0 OR TP_ZobrazHlasenieDoprNG_Plny = 0 THEN
		doMajak_ZlteSvetlo:= Blikac500ms;
	ELSE
		doMajak_ZlteSvetlo:= FALSE;
	END_IF

	//**********************************Červené svetlo majáka***************************************************//
	IF NastalaPorucha THEN
		doMajak_CerveneSvetlo:= Blikac500ms;
	ELSE
		doMajak_CerveneSvetlo:= FALSE;
	END_IF

	//***********************************Zvuková signalizácia majáka*********************************************//
	IF EDGEPOS (NastalaPorucha = TRUE) THEN
		ZapniHukacku:= TRUE;
	END_IF

	IF ZapniHukacku THEN
		doMajak_Hukacka:= Blikac500ms;
	ELSE
		doMajak_Hukacka:= FALSE;
	END_IF

	IF NOT NastalaPorucha THEN
		ZapniHukacku:= FALSE;
	ELSIF VypnutieHukacky THEN
		ZapniHukacku:= FALSE;
	END_IF

	//*********************************Potvrdenie alarmu**********************************************************//
	IF PotvrdenieAlarmov THEN
		Motion[1].cmd.autoInicialization:= TRUE;
		Motion[2].cmd.autoInicialization:= TRUE;
		Motion[3].cmd.autoInicialization:= TRUE;
		Motion[4].cmd.autoInicialization:= TRUE;
		FM_Menic[1].Input.Command.Acknowledge:= TRUE;
		FM_Menic[2].Input.Command.Acknowledge:= TRUE;
		FM_Menic[3].Input.Command.Acknowledge:= TRUE;

		brsmemset(ADR(Alarmy),0,SIZEOF(Alarmy));
		NastalaPorucha:= FALSE;
		CasPotvrdeniaAlarmu.IN:= TRUE;
		PoruchaZdvihuRotora:= FALSE;
		PoruchaOddelovaca:= FALSE;
		PoruchaOtocnyStol:= FALSE;
		PoruchaStanicaMerania:= FALSE;
		PoruchaStanicaRazenia:= FALSE;
		PoruchaStanicaStrihania:= FALSE;
		PoruchaStanicaValcovania:= FALSE;
		PoruchaStanicaValcovania2:= FALSE;
		PoruchaVstupManipulator:= FALSE;
		PoruchaVystupManipulator:= FALSE;
		PoruchaVystupOdsuvac:= FALSE;
		VypnutieHukacky:= TRUE;
		PotvrdenieAlarmov:= FALSE;
	END_IF

	IF CasPotvrdeniaAlarmu.Q AND Motion[1].errorID = 0 AND Motion[2].errorID = 0 AND Motion[3].errorID = 0 AND Motion[4].errorID = 0  THEN
		Motion[1].cmd.autoInicialization:= FALSE;
		Motion[2].cmd.autoInicialization:= FALSE;
		Motion[3].cmd.autoInicialization:= FALSE;
		Motion[4].cmd.autoInicialization:= FALSE;
		FM_Menic[1].Input.Command.Acknowledge:= FALSE;
		FM_Menic[2].Input.Command.Acknowledge:= FALSE;
		FM_Menic[3].Input.Command.Acknowledge:= FALSE;
		VypnutieHukacky:= FALSE;
		CasPotvrdeniaAlarmu.IN:= FALSE;
	END_IF

	CasPotvrdeniaAlarmu.PT:= T#2s;
	CasPotvrdeniaAlarmu();

	//******************************Porucha modulu DB1***********************************************************//
	IF SafetyPLC_Nabehlo AND NOT Modul_DB1_OK THEN
		Alarmy[92]:= TRUE;
	END_IF

	//******************************Porucha modulu DB2***********************************************************//
	IF SafetyPLC_Nabehlo AND NOT Modul_DB2_OK THEN
		Alarmy[93]:= TRUE;
	END_IF

	//******************************Porucha modulu DB3***********************************************************//
	IF SafetyPLC_Nabehlo AND NOT Modul_DB3_OK THEN
		Alarmy[94]:= TRUE;
	END_IF

	//******************************Porucha modulu DB4***********************************************************//
	IF SafetyPLC_Nabehlo AND NOT Modul_DB4_OK THEN
		Alarmy[95]:= TRUE;
	END_IF

	//******************************Porucha modulu DB5***********************************************************//
	IF SafetyPLC_Nabehlo AND NOT Modul_DB5_OK THEN
		Alarmy[96]:= TRUE;
	END_IF

	//******************************Porucha modulu DB6***********************************************************//
	IF SafetyPLC_Nabehlo AND NOT Modul_DB6_OK THEN
		Alarmy[97]:= TRUE;
	END_IF

	//******************************Porucha tlaku vzduchu*********************************************************//
	IF (Zariadenie_StavAutomat OR Zariadenie_StavManual) AND NOT diHlavnyPrivodVzduchu_TlakOK THEN
		Alarmy[0]:= TRUE;
	END_IF

	//******************************Stanica vonkajšieho valcovacia - Porucha tlaku vzduchu**********************************//
	IF Valcovanie2_Automat AND NOT diValc2_TlakPritlaku_OK THEN
		Alarmy[59]:= TRUE;
		PoruchaStanicaValcovania2:= TRUE;
	END_IF

	//******************************Bolo stlačené tlačítko CS*****************************************************//
	IF EDGENEG (Stav_CS_Odblokovane = TRUE) THEN
		Alarmy[1]:= TRUE;
	END_IF

	//*******************************Vstupný manipulátor - Porucha serva pojazdu**********************************************************************//
	IF (VstupManipulator_Automat OR VstupManipulator_Manual) AND Motion[1].error THEN
		Motion[1].cmd.halt:= TRUE;
		Alarmy[24]:= TRUE;
		PoruchaVstupManipulator:= TRUE;
	END_IF

	//*******************************Výstupný manipulátor - Porucha serva pojazdu**********************************************************************//
	IF (VystupManipulator_Automat OR VystupManipulator_Manual) AND Motion[2].error THEN
		Motion[2].cmd.halt:= TRUE;
		Alarmy[84]:= TRUE;
		PoruchaVystupManipulator:= TRUE;
	END_IF

	//*******************************Stanica vnútorného valcovania  - Porucha serva zdvihu nástroja**********************************************************************//
	IF (Valcovanie_Automat OR Valcovanie_Manual) AND Motion[3].error THEN
		Motion[3].cmd.halt:= TRUE;
		Alarmy[65]:= TRUE;
		PoruchaStanicaValcovania:= TRUE;
	END_IF

	//*******************************Stanica vonkajšieho valcovania  - Porucha serva zdvihu rotora**********************************************************************//
	IF (Valcovanie2_Automat OR Valcovanie2_Manual) AND Motion[4].error THEN
		Motion[4].cmd.halt:= TRUE;
		Alarmy[53]:= TRUE;
		PoruchaStanicaValcovania2:= TRUE;
	END_IF

	//**********************************Stanica merania - Porucha meniča *********************************************************************//
	IF (Meranie_Automat OR Meranie_Manual) AND (FM_Menic[1].Output.Status.Error OR NOT diMeranie_PoruchaOtacRotora) THEN
		Alarmy[72]:= TRUE;
		PoruchaStanicaMerania:= TRUE;
	END_IF

	//**********************************Stanica vnútorného valcovania - Porucha meniča *********************************************************************//
	IF (Valcovanie_Automat OR Valcovanie_Manual) AND (FM_Menic[2].Output.Status.Error OR NOT diValcovanie_PoruchaOtacRotora) THEN
		Alarmy[64]:= TRUE;
		PoruchaStanicaValcovania:= TRUE;
	END_IF

	//**********************************Stanica vonkajšieho valcovania - Porucha meniča *********************************************************************//
	IF (Valcovanie2_Automat OR Valcovanie2_Manual) AND (FM_Menic[3].Output.Status.Error OR NOT diValc2_PorMotoraOtacania) THEN
		Alarmy[54]:= TRUE;
		PoruchaStanicaValcovania2:= TRUE;
	END_IF

	//************************************Vstupný manipulátor - Pretazenie serva pojazdu************************************************************************//
	IF (VstupManipulator_Automat OR VstupManipulator_Manual) AND Motion[1].status.ActTorque > 1.7 THEN
		Motion[1].cmd.halt:= TRUE;
		Alarmy[25]:= TRUE;
		PoruchaVstupManipulator:= TRUE;
	END_IF

	//************************************Výstupný manipulátor - Pretazenie serva pojazdu************************************************************************//
	IF (VystupManipulator_Automat OR VystupManipulator_Manual) AND Motion[2].status.ActTorque > 1.7 THEN
		Motion[2].cmd.halt:= TRUE;
		Alarmy[85]:= TRUE;
		PoruchaVystupManipulator:= TRUE;
	END_IF

	//************************************Stanica vnútorného valcovania - Pretazenie serva zdvihu************************************************************************//
	IF (Valcovanie_Automat OR Valcovanie_Manual) AND Motion[3].status.ActTorque > 15.0 THEN
		Motion[3].cmd.halt:= TRUE;
		Alarmy[66]:= TRUE;
		PoruchaStanicaValcovania:= TRUE;
	END_IF

	//************************************Stanica vonkajšieho valcovania - Pretazenie serva zdvihu rotora************************************************************************//
	IF (Valcovanie2_Automat OR Valcovanie2_Manual) AND Motion[4].status.ActTorque > 15.0 THEN
		Motion[4].cmd.halt:= TRUE;
		Alarmy[55]:= TRUE;
		PoruchaStanicaValcovania2:= TRUE;
	END_IF

	//************************************Hydraulika - Nízka hladina oleja**************************************************************************************//
	IF NOT diHydraulika_HladinaOlejaOK THEN
		CasKontrolyOlejaHydrauliky.IN:= TRUE;
	ELSE
		CasKontrolyOlejaHydrauliky.IN:= FALSE;
	END_IF

	IF (Strihanie_Automat OR Razenie_Automat OR Strihanie_Manual OR Razenie_Manual) AND CasKontrolyOlejaHydrauliky.Q THEN
		Alarmy[2]:= TRUE;
		doHydraulika_ChodCerpadla:= FALSE;
		PoruchaStanicaRazenia:= TRUE;
		PoruchaStanicaStrihania:= TRUE;
	END_IF

	CasKontrolyOlejaHydrauliky.PT:= T#5s;
	CasKontrolyOlejaHydrauliky();

	//************************************Hydraulika - Porucha motora čerpadla***********************************************************************************//
	IF (Strihanie_Automat OR Razenie_Automat OR Strihanie_Manual OR Razenie_Manual) AND NOT diHydraulika_PoruchaCerpadla THEN
		Alarmy[3]:= TRUE;
		doHydraulika_ChodCerpadla:= FALSE;
		PoruchaStanicaRazenia:= TRUE;
		PoruchaStanicaStrihania:= TRUE;
	END_IF

//	************************************Hydraulika - Vysoká teplota oleja***********************************************************************************//
	IF (Strihanie_Automat OR Razenie_Automat OR Strihanie_Manual OR Razenie_Manual) AND NOT diHydraulika_TeplotaOlejaOK THEN
		Alarmy[4]:= TRUE;
		doHydraulika_ChodCerpadla:= FALSE;
		PoruchaStanicaRazenia:= TRUE;
		PoruchaStanicaStrihania:= TRUE;
	END_IF

	//************************************Hydraulika - Zanesenie olejového filtra***********************************************************************************//
	IF (Strihanie_Automat OR Razenie_Automat OR Strihanie_Manual OR Razenie_Manual) AND diHydraulika_Stav_FilterZaneseny THEN
		Alarmy[5]:= TRUE;
		doHydraulika_ChodCerpadla:= FALSE;
		PoruchaStanicaRazenia:= TRUE;
		PoruchaStanicaStrihania:= TRUE;
	END_IF

	//****************************************Otočný stol - porucha motora*****************************************************************************************//
	IF (Stol_Automat OR Stol_Manual) AND NOT diStol_PoruchaOtacStola THEN
		Alarmy[30]:= TRUE;
		PoruchaOtocnyStol:= TRUE;
	END_IF

	//***************************************Otočný stol - vysoka teplota motora****************************************************************************************//
	IF (Stol_Automat OR Stol_Manual) AND diStol_TeplotaMotoraOK THEN
		Alarmy[32]:= TRUE;
		PoruchaOtocnyStol:= TRUE;
	END_IF

		END_PROGRAM

PROGRAM _EXIT
		(* Insert code here *)

		END_PROGRAM
```

#### Variables.var - Local variables
```iecst
VAR
	i : INT;
	CasPotvrdeniaAlarmu : TON;
	ZapniHukacku : BOOL;
	CasKontrolyOlejaHydrauliky : TON;
	CasPoAktivaciiOplotenia : TON;
END_VAR
```

### Program Logical/Program/RychleDeje (IEC)

#### Main.st - Init, cyclic, exit code
```iecst
PROGRAM _INIT
	(* Insert code here *)

END_PROGRAM

PROGRAM _CYCLIC

	//Válcovanie 2 - Ovládanie brzdy motora válcovacieho nástroja//
	IF diValc2_OdbrzdOtacNastrojaMenic THEN
		doValc2_BrzdaOtacNastroja:= TRUE;
	ELSIF diValc2_OdbrzdOtacNastrojaRuka THEN
		doValc2_BrzdaOtacNastroja:= TRUE;
	ELSE
		doValc2_BrzdaOtacNastroja:= FALSE;
	END_IF

	//Valcovanie 2 - Kontrola otáčania nástroja//
	IF (*Valcovanie2_Automat AND*) FM_Menic[3].Output.Status.Running THEN
		Valc2_CasKontrolyOtacaniaNastr.IN:= NOT diValc2_SnimacOtacaniaNastroja;
	ELSE
		Valc2_CasKontrolyOtacaniaNastr.IN:= FALSE;
	END_IF

	IF Valc2_CasKontrolyOtacaniaNastr.Q THEN
		Alarmy[76]:= TRUE;
		PoruchaStanicaValcovania2:= TRUE;
	END_IF

	Valc2_CasKontrolyOtacaniaNastr.PT:= T#2s;
	Valc2_CasKontrolyOtacaniaNastr();

END_PROGRAM

PROGRAM _EXIT
	(* Insert code here *)

END_PROGRAM
```

#### Variables.var - Local variables
```iecst
VAR
	Valc2_CasKontrolyOtacaniaNastr : TON;
END_VAR
```

### Program Logical/Komunikacia/KOM_HlavnaLinka (IEC)

#### Main.st - Init, cyclic, exit code
```iecst
PROGRAM _INIT
	(* Insert code here *)

END_PROGRAM

PROGRAM _CYCLIC

	ModBus_Input1;
	ModBus_Input2;
	ModBus_Input3;
	ModBus_Input4;
	ModBus_Input5;
	ModBus_Output1;
	ModBus_Output2;
	ModBus_Output3;
	ModBus_Output4;
	ModBus_Output5;

	ZvolenaUroven:= ModBus_Input1;

END_PROGRAM

PROGRAM _EXIT
	(* Insert code here *)

END_PROGRAM
```

### Program Logical/PrihlasovaciSystem/PrihlasovaciSystem (IEC)
